// TwinCAT 3 PLC project PLC1
// ProgramVersion: 3.1.4023.0
// libraries:
//   Tc2_Standard, * (Beckhoff Automation GmbH)
//   Tc2_System, * (Beckhoff Automation GmbH)
//   Tc2_Utilities, * (Beckhoff Automation GmbH)
//   Tc3_EventLogger, * (Beckhoff Automation GmbH)
//   Tc3_Module, * (Beckhoff Automation GmbH)
//   Alarms Library,0.1,Atlantis
//   EASME Library Files,0.1,Atlantis
//   VisuSymbols,3.5.10.0,System
// project tree:
//   Alarm System/DUTs/02_Pitch/Hydair Data/ E_HydairState.TcDUT (not stored), E_LATState.TcDUT (not stored), E_MainState.TcDUT, Hydair_Data_Rcv.TcDUT (not stored), Hydair_Data_Send.TcDUT, Hydair_Ram_DataType.TcDUT (not stored), J1939_Inputs.TcDUT, J1939_outputs.TcDUT, ST_LoadSysCtrl.TcDUT (not stored), VARTYPE_EXTCANQUEUE.TcDUT
//   Alarm System/DUTs/02_Pitch/ PLCStruct.TcDUT (not stored), stLoadData.TcDUT, ST_BladePositionsEncoder.TcDUT (not stored), ST_DataSetEntry.TcDUT (not stored)
//   Alarm System/DUTs/02_Pitch/Test Rig/ E_StreamState.TcDUT (not stored)
//   Alarm System/DUTs/A. Operation_Ver2.10/02_Alarm_Handling/Alarms/ E_AlarmGroups.TcDUT, E_AlarmNames.TcDUT (not stored), E_AlarmProgram.TcDUT, E_AlarmState.TcDUT (not stored), E_BrakeProgram.TcDUT (not stored), E_ResetMode.TcDUT, ST_AlarmStructure.TcDUT, ST_Alarm_State.TcDUT (not stored), ST_Alarm_State_Alias.TcDUT (not stored), ST_AliasAlarms.TcDUT, ST_ProcessVariables.TcDUT, ST_Repetition.TcDUT (not stored), ST_RepetitionArray.TcDUT (not stored)
//   Alarm System/DUTs/A. Operation_Ver2.10/02_Alarm_Handling/StausCodes/03   STATUSCODES/ ARR_ListOfStatuscodesToBeSent.TcDUT
//   Alarm System/DUTs/A. Operation_Ver2.10/02_Alarm_Handling/StausCodes/08  Logging %28Harddisk%29/_01  Status Logger Objects/Intern/ E_FileState_SC.TcDUT (not stored), ST_FileSetup_SC.TcDUT (not stored)
//   Alarm System/DUTs/A. Operation_Ver2.10/02_Alarm_Handling/StausCodes/08  Logging %28Harddisk%29/_02  Event Logger/Logger Objects/ E_DataType.TcDUT (not stored)
//   Alarm System/DUTs/ E_IniNames.TcDUT, E_PitchState.TcDUT (not stored), stSSB_TCSInterface.TcDUT (not stored), ST_EmailSend.TcDUT (not stored), ST_EP9224_in.TcDUT (not stored), ST_EP9224_InputChannel.TcDUT, ST_EP9224_InputDevice.TcDUT (not stored), ST_EP9224_out.TcDUT, ST_EP9224_OutputChannel.TcDUT (not stored), ST_EP9224_SlaveIn.TcDUT, ST_EP9224_SlaveOut.TcDUT
//   Alarm System/DUTs/Safety/ ST_SafetyGroupData.TcDUT (not stored), ST_SafetyGroupTag.TcDUT
//   Alarm System/GVLs/A. Operation/01_General/ AlarmArrays.TcGVL, ArrIni.TcGVL (not stored), ArrLastAlarms.TcGVL (not stored), GlobVar_GeneralLog_Privat.TcGVL, GlobVar_GeneralLog_Public.TcGVL (not stored), GlobVar_LibStatuscodeLogger_Privat.TcGVL, GlobVar_ToBeReplaced_Public.TcGVL (not stored), GVL_Static.TcGVL, Operation.TcGVL (not stored), ProgramVersions.TcGVL, TurbineData.TcGVL
//   Alarm System/GVLs/A. Operation/ Global_Variables.TcGVL (not stored)
//   Alarm System/GVLs/ GVL_EventLogger.TcGVL
//   Alarm System/POUs/02_Alarm_Handling/ FB_AlarmHandler.TcPOU, FB_AlarmResetAccessCtrl.TcPOU (excluded from build), FB_AlarmResets.TcPOU, FB_AnalogueAlarm.TcPOU, FB_BrakeProgPriority.TcPOU (not stored), FB_HeaderForLogging.TcPOU (excluded from build), FB_MakeLoggString.TcPOU (excluded from build), FB_SendEmail.TcPOU, FB_StatusCodeLogger.TcPOU (excluded from build), FB_WriteEventData.TcPOU (excluded from build), FB_WriteEventData_Day.TcPOU (excluded from build), PRG_MAIN_StatuscodeLogger.TcPOU (excluded from build), PRG_Systemtime.TcPOU (not stored), P_AlarmHandling.TcPOU, P_AlarmTable.TcPOU, P_MainStatesAlarmCtrl.TcPOU (not stored), P_ScadaAlarmsMapping.TcPOU
//   Alarm System/POUs/02_Alarm_Handling/StatusCodes/ MAIN_R.TcPOU (not stored), PRG_TranslatorVarNames.TcPOU
//   Alarm System/TC3 EventLogger/ AlarmWithCustomSourceInfo.TcPOU (excluded from build), MultipleAlarmCreation.TcPOU, OtherAlarmsWithCustomSource.TcPOU (excluded from build), P_EventLogger_TCSAlarms.TcPOU
//   Base/Devices/DUT/ stError_VFD.TcDUT, stHMIMotorisedCB.TcDUT
//   Base/Devices/POU/ fbMotorisedCB.TcPOU
//   Base/Example/GVL/ GVL_HMI.TcGVL
//   Base/Example/POU/ POU_TestBase.TcPOU
//   Base/General Control/POU/ FB_AlarmEventSet.TcPOU, FB_TagAlarmProps.TcPOU, FB_Interlock.TcPOU, FB_Permissive.TcPOU, FB_SystemRunControl.TcPOU
//   Base/IO/DUT/ stError_AnalogueInput.TcDUT, stError_AnalogueOutput.TcDUT, stHMI_AnalogueInput.TcDUT, stHMI_AnalogueOutput.TcDUT, stHMI_DigitalInput.TcDUT (not stored), stHMI_DigitalOutput.TcDUT, stIOSensorTypes.TcDUT
//   Base/IO/POU/ fbIO_AnalogueInput.TcPOU, fbIO_AnalogueOutput.TcPOU, fbIO_DigitalInput.TcPOU, fbIO_DigitalOutput.TcPOU
//   Base/General Control/DUT/ stHMI_Interlock.TcDUT, stHMI_Permissive.TcDUT (not stored), stHMI_SystemRunControl.TcDUT
//   Base/Process Control/DUT/ stStep.TcDUT (not stored)
//   Base/Process Control/POU/ fb1dLookup.TcPOU, fb2dLookup.TcPOU, fbPulser.TcPOU, fbRateCalc.TcPOU, fbStepSequencer.TcPOU, POU.TcPOU
//   Base/Resource/ fbHMIBit.TcPOU
//   Base/Valve Control/DUT/ stError_Valve.TcDUT, stHMI_ValveControl.TcDUT
//   Base/Valve Control/POU/ fbValve_Solenoid.TcPOU, fcHMIBit.TcPOU
//   / GlobalTextList.TcGTLO, MAIN.TcPOU, PlcTask.TcTTO, Visualization Manager.TcVMO (not stored)
//   VISUs/ Visualization.TcVIS, Vis_AnalogueOutput_Symbol.TcVIS, Vis_DigitalInput_1.TcVIS, Vis_DigitalInput_2.TcVIS, Vis_Interlock_base.TcVIS
// real-time tasks:
//   TASK PlcTask: cycle T#10ms, priority 20, ADS port 350

CONFIGURATION PLC1
    RESOURCE PLC ON TwinCAT3
        TASK PlcTask(INTERVAL := T#10ms, PRIORITY := 20);
        PROGRAM MAIN WITH PlcTask : MAIN;
    END_RESOURCE
END_CONFIGURATION

// ---- Alarm System/DUTs/02_Pitch/Hydair Data/E_MainState.TcDUT
TYPE E_MainState :		//Is this the machine main state or the Hydraulics system??
(
	STOP:=0,
	STARTING_HYDRAULICS:=1,
	HYDRAULICS_READY:=2,
	IN_OPERATION:=3,
	PASSIVE:=5,
	MANUAL:=6,
	SAFETY_TRIPPED:=7,
	SHUTDOWN:=8
);
END_TYPE

// ---- Alarm System/DUTs/02_Pitch/Hydair Data/Hydair_Data_Send.TcDUT
TYPE Hydair_Data_Send :
STRUCT
	rRam1_LoadDemand:REAL;
	rRam2_LoadDemand:REAL;

	uiLoadsControl:ST_LoadSysCtrl;
END_STRUCT
END_TYPE

// ---- Alarm System/DUTs/02_Pitch/Hydair Data/J1939_Inputs.TcDUT
TYPE J1939_Inputs :
STRUCT
	TxCounter  : UINT;
	RxCounter  : UINT;
	NoOfRxMessages   : UINT;
	RxMessage  : ARRAY [0..11] OF VARTYPE_EXTCANQUEUE;
(*	NodeState  : USINT;
	DiagFlag   : BOOL;*)
END_STRUCT
END_TYPE

// ---- Alarm System/DUTs/02_Pitch/Hydair Data/J1939_outputs.TcDUT
TYPE J1939_outputs :
STRUCT
	TxCounter : UINT;
	RxCounter   : UINT;
	NoOfTxMessages    : UINT;
	TxMessage  : ARRAY [0..1] OF VARTYPE_EXTCANQUEUE;
END_STRUCT
END_TYPE

// ---- Alarm System/DUTs/02_Pitch/Hydair Data/VARTYPE_EXTCANQUEUE.TcDUT
TYPE VARTYPE_EXTCANQUEUE:
STRUCT
	length: UINT;
	cobId: UDINT;
	rxData: ARRAY [0..7] OF USINT;
END_STRUCT
END_TYPE

// ---- Alarm System/DUTs/02_Pitch/stLoadData.TcDUT
TYPE stLoadData :
STRUCT
	sLoadID: STRING[30];
	rRig1_LoadDemand:REAL;
	rRig2_LoadDemand:REAL;
	rRig3_LoadDemand:REAL;
	rPitchAngleDemand:REAL;
	bStart:BOOL;
	bConnect:BOOL;
	bHeartbeat:BOOL;
END_STRUCT
END_TYPE

// ---- Alarm System/DUTs/A. Operation_Ver2.10/02_Alarm_Handling/Alarms/E_AlarmGroups.TcDUT
TYPE E_AlarmGroups :
(
	Operation := 1,
	Safety := 2,
	Converter := 3,
	Pitch := 4,
	Yaw := 5,
	Nacelle := 6,
	Generator := 7,
	Gearbox := 8,
	AuxPower := 9,
	Grid := 10,
	SCADA := 11,
	BearingLube := 12,
	SealLube := 13,
	WaterMgt := 14,
	Brake := 15
);
END_TYPE

// ---- Alarm System/DUTs/A. Operation_Ver2.10/02_Alarm_Handling/Alarms/E_AlarmProgram.TcDUT
TYPE E_AlarmProgram :
(
	NoAction			:=0,	(* Prg1 *)
	Email				:=1,	(* Prg2 *)
	SMS					:=2

);
END_TYPE

// ---- Alarm System/DUTs/A. Operation_Ver2.10/02_Alarm_Handling/Alarms/E_ResetMode.TcDUT
TYPE E_ResetMode :
(
	AUTO			:=0,	(* Automatic after delay *)
	MANU			:=1	(* Manual *)
);
END_TYPE

// ---- Alarm System/DUTs/A. Operation_Ver2.10/02_Alarm_Handling/Alarms/ST_AlarmStructure.TcDUT
TYPE ST_AlarmStructure :
STRUCT
	sName:STRING;
	a:BOOL;
	b:BOOL;
	Changed:BOOL;
	iGroup:INT;
	iSetDelay:DINT;					(* 100ms *)
	iSetDelayElapsed:DINT;			(* 100ms *)
	iResetDelay:DINT;				(* 100ms *)
	iResetDelayElapsed:DINT;		(*100ms*)
	eResetMode:E_ResetMode;
	eBrakeProgram:E_BrakeProgram;
	eAlarmProgram:E_AlarmProgram;
	Enable: BOOL;
	TimeOcc: TIMESTRUCT;			(* Added 040405 KKa *)
	sTimeOcc: STRING(24); (* New *)	(* Added 091130 KKa *)
	Comment:STRING(255);

	iRepetitionNumber: INT;
	iRepetitionPeriod: INT; 					(*Minutes*)
	bRepetitionLimitExceeded: BOOL;

	Param1:ST_Parameters;
	Param2:ST_Parameters;

	iState:UDINT;(* New *)		(* Alarm state Active / Acked *)
	sID:STRING(5);(* New *)
	sClearName:STRING(90);(* New *)
	Index:INT;(* New *)
	bScope:BOOL;(* New *)

	stProcessVariables:ST_ProcessVariables; (* New *)

END_STRUCT
END_TYPE

// ---- Alarm System/DUTs/A. Operation_Ver2.10/02_Alarm_Handling/Alarms/ST_AliasAlarms.TcDUT
TYPE ST_AliasAlarms :
STRUCT
	b : INT;
END_STRUCT
END_TYPE

// ---- Alarm System/DUTs/A. Operation_Ver2.10/02_Alarm_Handling/Alarms/ST_ProcessVariables.TcDUT
TYPE ST_ProcessVariables :
STRUCT
	fPower:REAL;
	fFlowSpeed:REAL;
	fGeneratorSpeed:REAL;
	fPitchAngle:REAL;
END_STRUCT
END_TYPE

// ---- Alarm System/DUTs/A. Operation_Ver2.10/02_Alarm_Handling/StausCodes/03   STATUSCODES/ARR_ListOfStatuscodesToBeSent.TcDUT
TYPE ARR_ListOfStatuscodesToBeSent :
STRUCT
	arrListOfStatuscodesToBeSent: 		ARRAY [1..50] OF STRING [120];
END_STRUCT
END_TYPE

// ---- Alarm System/DUTs/E_IniNames.TcDUT
TYPE E_IniNames :
(
ini_fOperStartUpCounterMax := 1,
ini_fAlgHeartbeatCounterLimit := 2,
ini_fConverterCompensationAngle := 3,
ini_fConverterDampingTorqueLimitFactor := 4,
ini_fConverterDrivetrainDampingFactor1 := 5,
ini_fConverterDrivetrainDampingFactor2 := 6,
ini_fConverterDrivetrainDampingFactor3 := 7,
ini_fConverterExitToStandbyTimeout := 8,
ini_fConverterHeartbeatDelayms := 9,
ini_fConverterLookupSpeedVal0 := 10,
ini_fConverterLookupSpeedVal2 := 11,
ini_fConverterLookupSpeedVal4 := 12,
ini_fConverterLookupSpeedVal6 := 13,
ini_fConverterLookupSpeedVal8 := 14,
ini_fConverterLookupTorqueVal0 := 15,
ini_fConverterLookupTorqueVal2 := 16,
ini_fConverterLookupTorqueVal4 := 17,
ini_fConverterLookupTorqueVal6 := 18,
ini_fConverterLookupTorqueVal8 := 19,
ini_fConverterMinimumSpeedToStandby := 20,
ini_fConverterReductionReleaseFrequency := 21,
ini_fConverterReductionStartFrequency := 22,
ini_fConverterReductionStopFrequency := 23,
ini_fFlowSpeedAboveRatedLUTLength := 24,
ini_fFlowSpeedBelowRatedLUTLength := 25,
ini_fFlowSpeedTransitionLUTLength := 26,
ini_fGearboxRotorSpeedMin := 27,
ini_fGenPulloutC := 28,
ini_fGenPulloutM := 29,
ini_fGenSpeedNoiseFloor := 30,
ini_fOperEbbTideHeadingSetpoint := 31,
ini_fOperFloodTideHeadingSetpoint := 32,
ini_fOperFlowCutIn := 33,
ini_fOperFlowCutOut := 34,
ini_fOperFlowRated := 35,
ini_fOperInhibitPcsStbyToProd := 36,
ini_fOperMaxRotorPosErr := 37,
ini_fOperMinGenSyncSpeedRpm := 38,
ini_fOperRatedGeneratorSpeed := 39,
ini_fOperRotorPosCtrlErrOK := 40,
ini_fOperRotorSpeedRadsToStop := 41,
ini_fOperRotorStaticSpeedErr := 42,
ini_fOperSpeedHSSDiscrepMarginRpm := 43,
ini_fOperSpeedHSStoPCSDiscrepMarginRpm := 44,
ini_fOperSpeedLSStoHSSDiscrepMarginRpm := 45,
ini_fOperSpeedNoOfTargets := 46,
ini_fOperTrundleDuration := 47,
ini_fRotorBoltPosition := 48,
ini_fRotorEncoderZeroToBlade1 := 49,
ini_fRotorGBInputShaftPickupAPosition := 50,
ini_fRotorGBInputShaftPickupBPosition := 51,
ini_fSafetyDisablePCSEStop2 := 52,
ini_fSafetyDisablePCSEStop3 := 53,
ini_fSafetyPitchToFeatherTimeLimit := 54,
ini_fSafetyRotorDecelTimeLimit := 55,
ini_fTurbineGearboxRatio := 56,
ini_fVsprFastShutdownSpeedVal0 := 57,
ini_fVsprFastShutdownSpeedVal1 := 58,
ini_fVsprFastShutdownSpeedVal2 := 59,
ini_fVsprFastShutdownSpeedVal3 := 60,
ini_fVsprFastShutdownSpeedVal4 := 61,
ini_fVsprFastShutdownTorqueVal0 := 62,
ini_fVsprFastShutdownTorqueVal1 := 63,
ini_fVsprFastShutdownTorqueVal2 := 64,
ini_fVsprFastShutdownTorqueVal3 := 65,
ini_fVsprFastShutdownTorqueVal4 := 66,
ini_fVsprGenSpeedAtSyncSpeedRequiredTime := 67,
ini_fVsprLowSpeedSyncSpeedRPM := 68,
ini_fVsprMaximumFinePitchDeg := 69,
ini_fVsprMaximumGeneratorTorque := 70,
	ini_fVsprMinimumFinePitchDeg := 71,
ini_fVsprOptimalModeGain := 72,
ini_fVsprPositiveFeatherAngleDeg := 73,
ini_fVsprSpeedSetpointRateLimitRPMpSec := 74,
ini_fVsprStartupMinimumPitchRateLimitDegPSec := 75,
ini_fVsprSteadyShaftPowerLimit := 76,
ini_fVsprSyncSpeedTolRPM := 77,
ini_fVsprTorqueLimitSpeedVal0 := 78,
ini_fVsprTorqueLimitSpeedVal1 := 79,
ini_fVsprTorqueLimitSpeedVal2 := 80,
ini_fVsprTorqueLimitSpeedVal3 := 81,
ini_fVsprTorqueLimitSpeedVal4 := 82,
ini_fVsprTorqueLimitTorqueVal0 := 83,
ini_fVsprTorqueLimitTorqueVal1 := 84,
ini_fVsprTorqueLimitTorqueVal2 := 85,
ini_fVsprTorqueLimitTorqueVal3 := 86,
ini_fVsprTorqueLimitTorqueVal4 := 87,
ini_fWaterMgtNacelleBilgeLevelDefault := 88,
ini_fWaterMgtNacelleBilgePumpOffLevel := 89,
ini_fWaterMgtNacelleBilgePumpOffTimeMin := 90,
ini_fWaterMgtNacelleBilgePumpOffTimeout := 91,
ini_fWaterMgtNacelleBilgePumpOnLevel := 92,
ini_fWaterMgtNacelleBilgePumpOnTimeout := 93
);
END_TYPE

// ---- Alarm System/DUTs/Safety/ST_SafetyGroupTag.TcDUT
TYPE ST_SafetyGroupTag :
STRUCT
	sTitle	:STRING(80);
	bOutputSAFE	:BOOL;
	bError	:BOOL;
	bRun	:BOOL;
END_STRUCT
END_TYPE

// ---- Alarm System/DUTs/ST_EP9224_InputChannel.TcDUT
TYPE ST_EP9224_InputChannel :
STRUCT
	bErrorUs 	: BOOL;
	bErrorUp 	: BOOL;
	bWarningUs	: BOOL;
	bWarningUp	: BOOL;
	bStatusUs 	: BOOL;
	bStatusUp 	: BOOL;
	bChannelError : BOOL;
	bErrorSumCurrent 	      : BOOL;
(* This takes up a bit too much space and isn't maped by LMC, so leave it for now
	nCurrentUs 		: INT;
	nCurrentUp 		: INT;
*)
END_STRUCT
END_TYPE

// ---- Alarm System/DUTs/ST_EP9224_out.TcDUT
TYPE ST_EP9224_out :
STRUCT
	stOutput : ARRAY [1..EP9224_NUM_CHANNELS] OF ST_EP9224_OutputChannel;
	bGlobalReset : BOOL;
END_STRUCT
END_TYPE

// ---- Alarm System/DUTs/ST_EP9224_SlaveIn.TcDUT
TYPE ST_EP9224_SlaveIn :
STRUCT
	nOutput	:ARRAY [1..EP9224_NUM_CHANNELS] OF BYTE;
END_STRUCT
END_TYPE

// ---- Alarm System/DUTs/ST_EP9224_SlaveOut.TcDUT
TYPE ST_EP9224_SlaveOut :
STRUCT
	nChannel :ARRAY [1..EP9224_NUM_CHANNELS] OF BYTE;
	nStatus	 :BYTE;
END_STRUCT
END_TYPE

// ---- Base/Devices/DUT/stError_VFD.TcDUT
TYPE stError_VFD :
STRUCT
	MotorProtectorTripped: BOOL; (*Motor Protector tripped*)
	LocalDisconnectOff: BOOL; (*Motor Local switch OFF*)
	ClutchTripped: BOOL; 	(*Clutch error*)
	NoContactorFeedback: BOOL; (*No feedback from motor contactor*)
	ContactorStillOn: BOOL; (*Contactor still ON*)
	NoSignalForward: BOOL; (*No SIGNAL Forward from VFD*)
	NoSignalReverse: BOOL; (*No SIGNAL Reverse from VFD*)
	MotorNotStopped: BOOL; (*Motor doesn't stop*)
	MaxFrequencyReached: BOOL; (*Max frequency reached*)
	Overcurrent: BOOL; (*VFD overcurrent*)
	MotorOverload: BOOL; (*Motor overload*)
	VFDOverload: BOOL; (*VFD overload*)
	GeneralFault: BOOL; (*VFD fault*)
	NoCoolingFanFeedback: BOOL; (*Cooling fan did not come on within 30 seconds*)
END_STRUCT
END_TYPE

// ---- Base/Devices/DUT/stHMIMotorisedCB.TcDUT
TYPE stHMIMotorisedCB :
STRUCT
	iMode: 			 INT;
	iErrorCode:		 INT;		
	iStatus	:		 INT;	
	bPB_ResetError:	 BOOL; (*Reset errors pushbutton*)
	bPBEN_ResetError:BOOL; (*Reset Error pushbutton enable*)
	bPBOpen: 		 BOOL; (*Pushbutton command open from HMI*)
	bPBClose:		 BOOL; (*Pushbutton command close from HMI*)
	bPBEN_Open:		 BOOL; (*Pushbuton enable open command from HMI*)
	bPBEN_Close: 	 BOOL; (*Pushbuton enable open command from HMI*)
	bSignalClosed:	 BOOL; (*MCB closed feedback*)
	bSignalOpened: 	 BOOL; (*MCB Opened feedback*)
	bCloseON:		 BOOL; (*Close command is ON*)
	bOpenON:		 BOOL; (*Open command is ON*)
	bError:			 BOOL; (*Error Status*)
	bInterlock: 	 BOOL;	(*MCB Interlocked*)
END_STRUCT
END_TYPE

// ---- Base/IO/DUT/stError_AnalogueInput.TcDUT
TYPE stError_AnalogueInput :
STRUCT
	LowLowAlarm:BOOL; 	(*Value below low low set point*)
	HighHighAlarm:BOOL; (*Value above high high set point*)
	Invalid:BOOL; 		(*Invalid input*)
END_STRUCT
END_TYPE

// ---- Base/IO/DUT/stError_AnalogueOutput.TcDUT
TYPE stError_AnalogueOutput :
STRUCT
	Out_Of_Range:BOOL;			//Input Value is outside range of Engineering Units
	Configuration_Error:BOOL;	//Engineering Units are not properly configured
END_STRUCT
END_TYPE

// ---- Base/IO/DUT/stHMI_AnalogueInput.TcDUT
TYPE stHMI_AnalogueInput :
STRUCT
	iMode:INT; 			(*Current mode*)
	iErrorCode: INT; 	(*Error code*)
	iStatus:INT; 		(*Overall HMI Status*)
	rActiveValue:REAL;	(* Used Value, Input OR Override*)
	rInputValue:REAL; 	(*Input Value*)
	rManualValue:REAL; 	(*Manual mode simulated value*)
	bPB_ResetError:BOOL;  (*Reset errors pushbutton*)
	bPBEN_ResetError:BOOL; (*Reset error pushbutton enabled*)
	bError:BOOL;
END_STRUCT
END_TYPE

// ---- Base/IO/DUT/stHMI_AnalogueOutput.TcDUT
TYPE stHMI_AnalogueOutput :
STRUCT
	iMode: 			INT;		//Current mode
	iErrorCode:		INT; 		//error code	
	rValue:			REAL;		//Output Value
	rManualValue:	REAL;		//Manual mode value
	rAutoValue:		REAL;		 //Auto Mode Value
	rEstopValue:	REAL;		//Estop condition custom value
	bPB_ResetError:	BOOL;		//Reset errors pushbutton
	bPBEN_ResetError:	BOOL;	//Reset error pushbutton enabled
	bError:	BOOL;				//Overall error
	bInterlock:	BOOL;	//Analogue output is interlocked
	iEstopFunction:INT;	//Enumerated value of E-Stop response constant
END_STRUCT
END_TYPE

// ---- Base/IO/DUT/stHMI_DigitalOutput.TcDUT
TYPE stHMI_DigitalOutput :
STRUCT
	iMode:INT;			(*Current mode*)
	bCommand: BOOL;		(*Output command status*)
	bCommandAuto:BOOL;	(*the output command from the PLC, ignoring manual overrides*)
	bInterlock:BOOL;	(*Digital output is interlocked*)
	bPB_On:BOOL;		(*Command on override pushbutton*)
	bPB_Off:BOOL;		(*Command off override pushbutton*)
	bPBEN_On:BOOL;		(*Command on override pushbutton enabled*)
	bPBEN_Off:BOOL;		(*Command off override pushbutton enabled*)
END_STRUCT
END_TYPE

// ---- Base/IO/DUT/stIOSensorTypes.TcDUT
{attribute 'qualified_only'}
{attribute 'strict'}
TYPE stIOSensorTypes :
(
	AI_4To20ma := 0,
	AI_PT100	:= 1,
	AI_0To10V	:=2,
	AI_0To5V	:=3
	
);
END_TYPE

// ---- Base/General Control/DUT/stHMI_Interlock.TcDUT
TYPE stHMI_Interlock :
STRUCT
	abInterlocks: ARRAY[1..16] OF BOOL;
	asInterlockNames: ARRAY[1..16] OF STRING[20];
	bInterlockOk:BOOL;
END_STRUCT
END_TYPE

// ---- Base/General Control/DUT/stHMI_SystemRunControl.TcDUT
TYPE stHMI_SystemRunControl :
STRUCT
	bRunning:BOOL; 	  (*System is running*)
	bPB_Start:BOOL;    (*Start command pushbutton*)
	bPB_Stop:BOOL;	  (*Stop command pushbutton*)
	bPBEN_Start:BOOL;  (*Start command pushbutton enable*)
	bPBEN_Stop:BOOL;  (*Stop command pushbutton enable*)
END_STRUCT
END_TYPE

// ---- Base/Valve Control/DUT/stError_Valve.TcDUT
TYPE stError_Valve :
STRUCT
	NoHomeFeedback:BOOL;			//Home position feedback not active
	NoWorkFeedback:BOOL;			//Work position feedback not active
	HomeFeedbackStillActive: BOOL;	//Home position feedback still active when commanded to Work Position
	WorkFeedbackStillActive: BOOL;	//Work position feedback still active when commanded to Home Position
END_STRUCT
END_TYPE

// ---- Base/Valve Control/DUT/stHMI_ValveControl.TcDUT
TYPE stHMI_ValveControl :
STRUCT
	iMode	:		 INT;		//Current mode				
	iErrorCode:		 INT;		//
	iStatus	:		 INT;		//
	bPB_ResetError:	 BOOL;		//Reset errors pushbutton
	bPB_Home:		 BOOL;		//Move to home in manual mode pushbutton
	bPB_Work:		 BOOL;		//Move to work in manual mode pushbutton
	bPBEN_ResetError:BOOL;		//Reset Error pushbutton enable
	bPBEN_Home:		 BOOL;		//Home pushbutton enabled
	bPBEN_Work:		 BOOL;		//Work pushbutton enabledv
	bHomeOn:		 BOOL;		//Home command is on
	bWorkOn:		 BOOL;		//Work command is on
	bSignalHome:	 BOOL;		//Home feedback
	bSignalWork:	 BOOL;		//Work feedback
	bError:			 BOOL;		//Error Status
	bInterlock: 	 BOOL;		//Valve Interlocked
END_STRUCT
END_TYPE

// ---- Alarm System/GVLs/A. Operation/01_General/AlarmArrays.TcGVL
{attribute 'Tc2GvlVarNames'}
VAR_GLOBAL
	{attribute 'OPC.UA.DA' := '1'}
	{attribute 'OPC.UA.DA.StructuredType' := '1'}
	arrScadaAlarms : ARRAY [1..222]  OF ST_AliasAlarms;	
	
	{attribute 'OPC.UA.DA' := '1'}
	{attribute 'OPC.UA.DA.StructuredType' := '1'}
	arrOPCUA_Alarms : ARRAY [1..10]  OF ST_Alarm_State_Alias;	
	
	
END_VAR


VAR_GLOBAL PERSISTENT
stOperAlarmIniFileName: STRING:='Alarms_AR2000.xls 011021';
arrAlarmsOld: ARRAY [1..222] OF ST_AlarmStructure;
arrAlarmsOriginal,arrAlarms: ARRAY [1..222] OF ST_AlarmStructure :=[
( sName := 'a_bOperMaStInitSt', sClearName := '', sID := '1001', a := FALSE, b := FALSE, iGroup :=1, iSetDelay :=0, iResetDelay := 100, eResetMode := MANU, eBrakeProgram := B100, eAlarmProgram := 0, Enable := TRUE, iRepetitionNumber := 0 , iRepetitionPeriod := 10, Comment := 'Turbine Initialising', Param1 := (Set:=0, SetMin:=0, SetMax:=0,Comment:=''), Param2 := (Set:=0, SetMin:=0, SetMax:=0,Comment:='') ),
( sName := 'a_bOperMaStStopSt', sClearName := '', sID := '1002', a := FALSE, b := FALSE, iGroup :=1, iSetDelay :=0, iResetDelay := 0, eResetMode := MANU, eBrakeProgram := B100, eAlarmProgram := 0, Enable := TRUE, iRepetitionNumber := 0 , iRepetitionPeriod := 10, Comment := 'Turbine in the Stop state', Param1 := (Set:=0, SetMin:=0, SetMax:=0,Comment:=''), Param2 := (Set:=0, SetMin:=0, SetMax:=0,Comment:='') ),
( sName := 'a_bOperMaStIdleSt', sClearName := '', sID := '1003', a := FALSE, b := FALSE, iGroup :=1, iSetDelay :=0, iResetDelay := 0, eResetMode := MANU, eBrakeProgram := B100, eAlarmProgram := 0, Enable := TRUE, iRepetitionNumber := 0 , iRepetitionPeriod := 10, Comment := 'Turbine in the Idle state', Param1 := (Set:=0, SetMin:=0, SetMax:=0,Comment:=''), Param2 := (Set:=0, SetMin:=0, SetMax:=0,Comment:='') ),
( sName := 'a_bOperMaStStandbySt', sClearName := '', sID := '1004', a := FALSE, b := FALSE, iGroup :=1, iSetDelay :=0, iResetDelay := 0, eResetMode := MANU, eBrakeProgram := B100, eAlarmProgram := 0, Enable := TRUE, iRepetitionNumber := 0 , iRepetitionPeriod := 10, Comment := 'Turbine in the Ready state', Param1 := (Set:=0, SetMin:=0, SetMax:=0,Comment:=''), Param2 := (Set:=0, SetMin:=0, SetMax:=0,Comment:='') ),
( sName := 'a_bOperMaStPowerProductionSt', sClearName := '', sID := '1005', a := FALSE, b := FALSE, iGroup :=1, iSetDelay :=0, iResetDelay := 0, eResetMode := MANU, eBrakeProgram := B100, eAlarmProgram := 0, Enable := TRUE, iRepetitionNumber := 0 , iRepetitionPeriod := 10, Comment := 'Turbine in the Power Production state', Param1 := (Set:=0, SetMin:=0, SetMax:=0,Comment:=''), Param2 := (Set:=0, SetMin:=0, SetMax:=0,Comment:='') ),
( sName := 'a_bOperMaStNormalStopSt', sClearName := '', sID := '1006', a := FALSE, b := FALSE, iGroup :=1, iSetDelay :=0, iResetDelay := 0, eResetMode := MANU, eBrakeProgram := B100, eAlarmProgram := 0, Enable := TRUE, iRepetitionNumber := 0 , iRepetitionPeriod := 10, Comment := 'Turbine in the Normal Stop state', Param1 := (Set:=0, SetMin:=0, SetMax:=0,Comment:=''), Param2 := (Set:=0, SetMin:=0, SetMax:=0,Comment:='') ),
( sName := 'a_bOperMaStEmergencyStopSt', sClearName := '', sID := '1007', a := FALSE, b := FALSE, iGroup :=1, iSetDelay :=0, iResetDelay := 0, eResetMode := MANU, eBrakeProgram := B100, eAlarmProgram := 0, Enable := TRUE, iRepetitionNumber := 0 , iRepetitionPeriod := 10, Comment := 'Turbine in the Emergency Stop state', Param1 := (Set:=0, SetMin:=0, SetMax:=0,Comment:=''), Param2 := (Set:=0, SetMin:=0, SetMax:=0,Comment:='') ),
( sName := 'a_bOperAutostartCmdActive', sClearName := '', sID := '1008', a := FALSE, b := FALSE, iGroup :=1, iSetDelay :=0, iResetDelay := 0, eResetMode := MANU, eBrakeProgram := B99, eAlarmProgram := 0, Enable := TRUE, iRepetitionNumber := 0 , iRepetitionPeriod := 0, Comment := 'System generation inhibit removed by operator', Param1 := (Set:=0, SetMin:=0, SetMax:=0,Comment:=''), Param2 := (Set:=0, SetMin:=0, SetMax:=0,Comment:='') ),
( sName := 'a_bOperTestIdlingShutdown', sClearName := '', sID := '1009', a := FALSE, b := FALSE, iGroup :=1, iSetDelay :=0, iResetDelay := 0, eResetMode := MANU, eBrakeProgram := B17, eAlarmProgram := 0, Enable := TRUE, iRepetitionNumber := 0 , iRepetitionPeriod := 0, Comment := 'Test B17 go to Idle or Standby', Param1 := (Set:=0, SetMin:=0, SetMax:=0,Comment:=''), Param2 := (Set:=0, SetMin:=0, SetMax:=0,Comment:='') ),
( sName := 'a_bOperTestBrakingShutdown', sClearName := '', sID := '1010', a := FALSE, b := FALSE, iGroup :=1, iSetDelay :=0, iResetDelay := 0, eResetMode := MANU, eBrakeProgram := B14, eAlarmProgram := 0, Enable := TRUE, iRepetitionNumber := 0 , iRepetitionPeriod := 0, Comment := 'Test B14 apply parking brake', Param1 := (Set:=0, SetMin:=0, SetMax:=0,Comment:=''), Param2 := (Set:=0, SetMin:=0, SetMax:=0,Comment:='') ),
( sName := 'a_bOperTestSafetyVCTripShutdown', sClearName := '', sID := '1011', a := FALSE, b := FALSE, iGroup :=1, iSetDelay :=0, iResetDelay := 0, eResetMode := MANU, eBrakeProgram := B100, eAlarmProgram := 0, Enable := TRUE, iRepetitionNumber := 0 , iRepetitionPeriod := 0, Comment := 'Test B9 trip vacuum contactor', Param1 := (Set:=0, SetMin:=0, SetMax:=0,Comment:=''), Param2 := (Set:=0, SetMin:=0, SetMax:=0,Comment:='') ),
( sName := 'a_bOperTestSafetyBrakeShutdown', sClearName := '', sID := '1012', a := FALSE, b := FALSE, iGroup :=1, iSetDelay :=0, iResetDelay := 0, eResetMode := MANU, eBrakeProgram := B100, eAlarmProgram := 0, Enable := TRUE, iRepetitionNumber := 0 , iRepetitionPeriod := 0, Comment := 'Test B5 apply safety brake', Param1 := (Set:=0, SetMin:=0, SetMax:=0,Comment:=''), Param2 := (Set:=0, SetMin:=0, SetMax:=0,Comment:='') ),
( sName := 'a_bOperCmdNormalShutdownToStop', sClearName := 'Turbine manual stop using main gui button', sID := '1013', a := FALSE, b := FALSE, iGroup :=1, iSetDelay :=0, iResetDelay := 0, eResetMode := MANU, eBrakeProgram := B100, eAlarmProgram := 0, Enable := TRUE, iRepetitionNumber := 0 , iRepetitionPeriod := 0, Comment := 'Manual stop command', Param1 := (Set:=0, SetMin:=0, SetMax:=0,Comment:=''), Param2 := (Set:=0, SetMin:=0, SetMax:=0,Comment:='') ),
( sName := 'a_bOperCmdNormalShutdownToStandby', sClearName := '', sID := '1014', a := FALSE, b := FALSE, iGroup :=1, iSetDelay :=0, iResetDelay := 0, eResetMode := MANU, eBrakeProgram := B100, eAlarmProgram := 0, Enable := TRUE, iRepetitionNumber := 0 , iRepetitionPeriod := 0, Comment := '', Param1 := (Set:=0, SetMin:=0, SetMax:=0,Comment:=''), Param2 := (Set:=0, SetMin:=0, SetMax:=0,Comment:='') ),
( sName := 'a_bOperRepeatingAlarm', sClearName := '', sID := '1015', a := FALSE, b := FALSE, iGroup :=1, iSetDelay :=10, iResetDelay := 0, eResetMode := MANU, eBrakeProgram := B100, eAlarmProgram := 0, Enable := TRUE, iRepetitionNumber := 0 , iRepetitionPeriod := 10, Comment := 'Alarm which occur with this one has occured too many times', Param1 := (Set:=0, SetMin:=0, SetMax:=0,Comment:=''), Param2 := (Set:=0, SetMin:=0, SetMax:=0,Comment:='') ),
( sName := 'a_bOperResetTooLongPushed', sClearName := 'Reset Button ', sID := '1016', a := FALSE, b := FALSE, iGroup :=1, iSetDelay :=10, iResetDelay := 0, eResetMode := MANU, eBrakeProgram := B99, eAlarmProgram := 0, Enable := TRUE, iRepetitionNumber := 0 , iRepetitionPeriod := 10, Comment := 'Reset button pressed too long', Param1 := (Set:=0, SetMin:=0, SetMax:=0,Comment:=''), Param2 := (Set:=0, SetMin:=0, SetMax:=0,Comment:='') ),
( sName := 'a_bOperAlarmParameterChanged', sClearName := 'Alarm Parameter ', sID := '1017', a := FALSE, b := FALSE, iGroup :=1, iSetDelay :=0, iResetDelay := 5, eResetMode := MANU, eBrakeProgram := B99, eAlarmProgram := 0, Enable := TRUE, iRepetitionNumber := 0 , iRepetitionPeriod := 10, Comment := 'Alarm parameter has been changed', Param1 := (Set:=0, SetMin:=0, SetMax:=0,Comment:=''), Param2 := (Set:=0, SetMin:=0, SetMax:=0,Comment:='') ),
( sName := 'a_bOperIniParameterChanged', sClearName := 'Ini Parameter ', sID := '1018', a := FALSE, b := FALSE, iGroup :=1, iSetDelay :=0, iResetDelay := 5, eResetMode := MANU, eBrakeProgram := B99, eAlarmProgram := 0, Enable := TRUE, iRepetitionNumber := 0 , iRepetitionPeriod := 10, Comment := 'Ini parameter has been changed', Param1 := (Set:=0, SetMin:=0, SetMax:=0,Comment:=''), Param2 := (Set:=0, SetMin:=0, SetMax:=0,Comment:='') ),
( sName := 'a_bOperSystemReboot', sClearName := 'System ', sID := '1019', a := FALSE, b := FALSE, iGroup :=1, iSetDelay :=10, iResetDelay := 150, eResetMode := MANU, eBrakeProgram := B100, eAlarmProgram := 0, Enable := TRUE, iRepetitionNumber := 0 , iRepetitionPeriod := 10, Comment := 'System is rebooted', Param1 := (Set:=0, SetMin:=0, SetMax:=0,Comment:=''), Param2 := (Set:=0, SetMin:=0, SetMax:=0,Comment:='') ),
( sName := 'a_bOperSystemRestart ', sClearName := 'System ', sID := '1020', a := FALSE, b := FALSE, iGroup :=1, iSetDelay :=10, iResetDelay := 150, eResetMode := MANU, eBrakeProgram := B100, eAlarmProgram := 0, Enable := TRUE, iRepetitionNumber := 0 , iRepetitionPeriod := 10, Comment := 'System is restarted', Param1 := (Set:=0, SetMin:=0, SetMax:=0,Comment:=''), Param2 := (Set:=0, SetMin:=0, SetMax:=0,Comment:='') ),
( sName := 'a_bOperScopeViewNotActive', sClearName := 'ScopeView running', sID := '1021', a := FALSE, b := FALSE, iGroup :=1, iSetDelay :=100, iResetDelay := 0, eResetMode := MANU, eBrakeProgram := B17, eAlarmProgram := 0, Enable := TRUE, iRepetitionNumber := 0 , iRepetitionPeriod := 10, Comment := 'Fastlog system not active', Param1 := (Set:=0, SetMin:=0, SetMax:=0,Comment:=''), Param2 := (Set:=0, SetMin:=0, SetMax:=0,Comment:='') ),
( sName := 'a_bOperXMLDataUncertainty', sClearName := 'Turbine data XML file Ok', sID := '1022', a := FALSE, b := FALSE, iGroup :=1, iSetDelay :=0, iResetDelay := 0, eResetMode := MANU, eBrakeProgram := B17, eAlarmProgram := 0, Enable := TRUE, iRepetitionNumber := 0 , iRepetitionPeriod := 10, Comment := 'Turbine data XML file uncertainty', Param1 := (Set:=0, SetMin:=0, SetMax:=0,Comment:=''), Param2 := (Set:=0, SetMin:=0, SetMax:=0,Comment:='') ),
( sName := 'a_bOperSoftwareUpdate', sClearName := 'System software ', sID := '1023', a := FALSE, b := FALSE, iGroup :=1, iSetDelay :=0, iResetDelay := 0, eResetMode := MANU, eBrakeProgram := B17, eAlarmProgram := 0, Enable := FALSE, iRepetitionNumber := 0 , iRepetitionPeriod := 10, Comment := 'System software is updated', Param1 := (Set:=0, SetMin:=0, SetMax:=0,Comment:=''), Param2 := (Set:=0, SetMin:=0, SetMax:=0,Comment:='') ),
( sName := 'a_bOperFastlogComsErr', sClearName := 'a_bOperLossOfCommsToArrayController', sID := '1024', a := FALSE, b := FALSE, iGroup :=1, iSetDelay :=0, iResetDelay := 0, eResetMode := MANU, eBrakeProgram := B99, eAlarmProgram := 0, Enable := TRUE, iRepetitionNumber := 0 , iRepetitionPeriod := 10, Comment := 'Loss of Comms with ARL Array PLC', Param1 := (Set:=0, SetMin:=0, SetMax:=0,Comment:=''), Param2 := (Set:=0, SetMin:=0, SetMax:=0,Comment:='') ),
( sName := 'a_bOperInOffMode', sClearName := 'Turbine in OFF Mode', sID := '1025', a := FALSE, b := FALSE, iGroup :=1, iSetDelay :=0, iResetDelay := 0, eResetMode := MANU, eBrakeProgram := B100, eAlarmProgram := 0, Enable := TRUE, iRepetitionNumber := 0 , iRepetitionPeriod := 10, Comment := 'Turbine entering OFF Mode', Param1 := (Set:=0, SetMin:=0, SetMax:=0,Comment:=''), Param2 := (Set:=0, SetMin:=0, SetMax:=0,Comment:='') ),
( sName := 'a_bOperInServiceMode', sClearName := 'Turbine in Service Mode', sID := '1026', a := FALSE, b := FALSE, iGroup :=1, iSetDelay :=0, iResetDelay := 0, eResetMode := MANU, eBrakeProgram := B100, eAlarmProgram := 0, Enable := TRUE, iRepetitionNumber := 0 , iRepetitionPeriod := 10, Comment := 'Turbine entering Service Mode', Param1 := (Set:=0, SetMin:=0, SetMax:=0,Comment:=''), Param2 := (Set:=0, SetMin:=0, SetMax:=0,Comment:='') ),
( sName := 'a_bOperInAutomaticMode', sClearName := 'Turbine in Automatic Mode', sID := '1027', a := FALSE, b := FALSE, iGroup :=1, iSetDelay :=0, iResetDelay := 0, eResetMode := MANU, eBrakeProgram := B100, eAlarmProgram := 0, Enable := TRUE, iRepetitionNumber := 0 , iRepetitionPeriod := 10, Comment := 'Turbine entering Automatic Mode', Param1 := (Set:=0, SetMin:=0, SetMax:=0,Comment:=''), Param2 := (Set:=0, SetMin:=0, SetMax:=0,Comment:='') ),
( sName := 'a_bOperInManualMode', sClearName := 'Turbine in Manual Mode', sID := '1028', a := FALSE, b := FALSE, iGroup :=1, iSetDelay :=0, iResetDelay := 0, eResetMode := MANU, eBrakeProgram := B100, eAlarmProgram := 0, Enable := TRUE, iRepetitionNumber := 0 , iRepetitionPeriod := 10, Comment := 'Turbine entering Manual Mode', Param1 := (Set:=0, SetMin:=0, SetMax:=0,Comment:=''), Param2 := (Set:=0, SetMin:=0, SetMax:=0,Comment:='') ),
( sName := 'a_bOperInFATMode', sClearName := 'Turbine in Factory Acceptance Test Nautilus Mode', sID := '1029', a := FALSE, b := FALSE, iGroup :=1, iSetDelay :=0, iResetDelay := 0, eResetMode := MANU, eBrakeProgram := B100, eAlarmProgram := 0, Enable := TRUE, iRepetitionNumber := 0 , iRepetitionPeriod := 10, Comment := 'Turbine entering Factory Acceptance Test Nautilus Mode', Param1 := (Set:=0, SetMin:=0, SetMax:=0,Comment:=''), Param2 := (Set:=0, SetMin:=0, SetMax:=0,Comment:='') ),
( sName := 'a_bHydairFaultActive', sClearName := 'Cleared', sID := '1030', a := FALSE, b := FALSE, iGroup :=1, iSetDelay :=0, iResetDelay := 0, eResetMode := MANU, eBrakeProgram := B99, eAlarmProgram := 0, Enable := TRUE, iRepetitionNumber := 0 , iRepetitionPeriod := 0, Comment := '', Param1 := (Set:=0, SetMin:=0, SetMax:=0,Comment:=''), Param2 := (Set:=0, SetMin:=0, SetMax:=0,Comment:='') ),
( sName := 'a_bHydairOfflineFilterClogged', sClearName := 'Cleared', sID := '1031', a := FALSE, b := FALSE, iGroup :=1, iSetDelay :=0, iResetDelay := 0, eResetMode := MANU, eBrakeProgram := B99, eAlarmProgram := 0, Enable := TRUE, iRepetitionNumber := 0 , iRepetitionPeriod := 0, Comment := '', Param1 := (Set:=0, SetMin:=0, SetMax:=0,Comment:=''), Param2 := (Set:=0, SetMin:=0, SetMax:=0,Comment:='') ),
( sName := 'a_bMainReturnPressureFilterClogged', sClearName := 'Cleared', sID := '1032', a := FALSE, b := FALSE, iGroup :=1, iSetDelay :=0, iResetDelay := 0, eResetMode := MANU, eBrakeProgram := B99, eAlarmProgram := 0, Enable := TRUE, iRepetitionNumber := 0 , iRepetitionPeriod := 0, Comment := '', Param1 := (Set:=0, SetMin:=0, SetMax:=0,Comment:=''), Param2 := (Set:=0, SetMin:=0, SetMax:=0,Comment:='') ),
( sName := 'a_bMainSupplyPressureFilterClogged', sClearName := 'Cleared', sID := '1033', a := FALSE, b := FALSE, iGroup :=1, iSetDelay :=0, iResetDelay := 0, eResetMode := MANU, eBrakeProgram := B99, eAlarmProgram := 0, Enable := TRUE, iRepetitionNumber := 0 , iRepetitionPeriod := 0, Comment := '', Param1 := (Set:=0, SetMin:=0, SetMax:=0,Comment:=''), Param2 := (Set:=0, SetMin:=0, SetMax:=0,Comment:='') ),
( sName := 'a_bHydairPassiveCtrlState', sClearName := 'Cleared', sID := '1034', a := FALSE, b := FALSE, iGroup :=1, iSetDelay :=0, iResetDelay := 0, eResetMode := MANU, eBrakeProgram := B99, eAlarmProgram := 0, Enable := TRUE, iRepetitionNumber := 0 , iRepetitionPeriod := 0, Comment := '', Param1 := (Set:=0, SetMin:=0, SetMax:=0,Comment:=''), Param2 := (Set:=0, SetMin:=0, SetMax:=0,Comment:='') ),
( sName := 'a_bHydairStartUp', sClearName := 'Cleared', sID := '1035', a := FALSE, b := FALSE, iGroup :=1, iSetDelay :=0, iResetDelay := 0, eResetMode := MANU, eBrakeProgram := B99, eAlarmProgram := 0, Enable := TRUE, iRepetitionNumber := 0 , iRepetitionPeriod := 0, Comment := '', Param1 := (Set:=0, SetMin:=0, SetMax:=0,Comment:=''), Param2 := (Set:=0, SetMin:=0, SetMax:=0,Comment:='') ),
( sName := 'a_bHydairReadyToOperate', sClearName := 'Cleared', sID := '1036', a := FALSE, b := FALSE, iGroup :=1, iSetDelay :=0, iResetDelay := 0, eResetMode := MANU, eBrakeProgram := B99, eAlarmProgram := 0, Enable := TRUE, iRepetitionNumber := 0 , iRepetitionPeriod := 0, Comment := '', Param1 := (Set:=0, SetMin:=0, SetMax:=0,Comment:=''), Param2 := (Set:=0, SetMin:=0, SetMax:=0,Comment:='') ),
( sName := 'a_bHydairActiveCtrlState', sClearName := 'Cleared', sID := '1037', a := FALSE, b := FALSE, iGroup :=1, iSetDelay :=0, iResetDelay := 0, eResetMode := MANU, eBrakeProgram := B99, eAlarmProgram := 0, Enable := TRUE, iRepetitionNumber := 0 , iRepetitionPeriod := 0, Comment := '', Param1 := (Set:=0, SetMin:=0, SetMax:=0,Comment:=''), Param2 := (Set:=0, SetMin:=0, SetMax:=0,Comment:='') ),
( sName := 'a_bHydairStopped', sClearName := 'Cleared', sID := '1038', a := FALSE, b := FALSE, iGroup :=1, iSetDelay :=0, iResetDelay := 0, eResetMode := MANU, eBrakeProgram := B99, eAlarmProgram := 0, Enable := TRUE, iRepetitionNumber := 0 , iRepetitionPeriod := 0, Comment := '', Param1 := (Set:=0, SetMin:=0, SetMax:=0,Comment:=''), Param2 := (Set:=0, SetMin:=0, SetMax:=0,Comment:='') ),
( sName := 'a_bHydairEstopActive', sClearName := 'Cleared', sID := '1039', a := FALSE, b := FALSE, iGroup :=1, iSetDelay :=0, iResetDelay := 0, eResetMode := MANU, eBrakeProgram := B99, eAlarmProgram := 0, Enable := TRUE, iRepetitionNumber := 0 , iRepetitionPeriod := 0, Comment := '', Param1 := (Set:=0, SetMin:=0, SetMax:=0,Comment:=''), Param2 := (Set:=0, SetMin:=0, SetMax:=0,Comment:='') ),
( sName := 'a_bHydairOilTempTooHigh', sClearName := 'Cleared', sID := '1040', a := FALSE, b := FALSE, iGroup :=1, iSetDelay :=0, iResetDelay := 0, eResetMode := MANU, eBrakeProgram := B99, eAlarmProgram := 0, Enable := TRUE, iRepetitionNumber := 0 , iRepetitionPeriod := 0, Comment := '', Param1 := (Set:=0, SetMin:=0, SetMax:=0,Comment:=''), Param2 := (Set:=0, SetMin:=0, SetMax:=0,Comment:='') ),
( sName := 'a_bHydairReadyToStartup', sClearName := 'Cleared', sID := '1041', a := FALSE, b := FALSE, iGroup :=1, iSetDelay :=0, iResetDelay := 0, eResetMode := MANU, eBrakeProgram := B99, eAlarmProgram := 0, Enable := TRUE, iRepetitionNumber := 0 , iRepetitionPeriod := 0, Comment := '', Param1 := (Set:=0, SetMin:=0, SetMax:=0,Comment:=''), Param2 := (Set:=0, SetMin:=0, SetMax:=0,Comment:='') ),
( sName := 'a_bOperRequestStopLATSystem', sClearName := 'Cleared', sID := '1042', a := FALSE, b := FALSE, iGroup :=1, iSetDelay :=0, iResetDelay := 0, eResetMode := MANU, eBrakeProgram := B99, eAlarmProgram := 0, Enable := TRUE, iRepetitionNumber := 0 , iRepetitionPeriod := 0, Comment := '', Param1 := (Set:=0, SetMin:=0, SetMax:=0,Comment:=''), Param2 := (Set:=0, SetMin:=0, SetMax:=0,Comment:='') ),
( sName := 'a_bOperRequestStartupHydair', sClearName := 'Cleared', sID := '1043', a := FALSE, b := FALSE, iGroup :=1, iSetDelay :=0, iResetDelay := 0, eResetMode := MANU, eBrakeProgram := B99, eAlarmProgram := 0, Enable := TRUE, iRepetitionNumber := 0 , iRepetitionPeriod := 0, Comment := '', Param1 := (Set:=0, SetMin:=0, SetMax:=0,Comment:=''), Param2 := (Set:=0, SetMin:=0, SetMax:=0,Comment:='') ),
( sName := 'a_bOperRequestPassivePitchCtrl', sClearName := 'Cleared', sID := '1044', a := FALSE, b := FALSE, iGroup :=1, iSetDelay :=0, iResetDelay := 0, eResetMode := MANU, eBrakeProgram := B99, eAlarmProgram := 0, Enable := TRUE, iRepetitionNumber := 0 , iRepetitionPeriod := 0, Comment := '', Param1 := (Set:=0, SetMin:=0, SetMax:=0,Comment:=''), Param2 := (Set:=0, SetMin:=0, SetMax:=0,Comment:='') ),
( sName := 'a_bOperRequestActiveLoadCtrlMode', sClearName := 'Cleared', sID := '1045', a := FALSE, b := FALSE, iGroup :=1, iSetDelay :=0, iResetDelay := 0, eResetMode := MANU, eBrakeProgram := B99, eAlarmProgram := 0, Enable := TRUE, iRepetitionNumber := 0 , iRepetitionPeriod := 0, Comment := '', Param1 := (Set:=0, SetMin:=0, SetMax:=0,Comment:=''), Param2 := (Set:=0, SetMin:=0, SetMax:=0,Comment:='') ),
( sName := 'a_bOperRequestLoadProfileStream', sClearName := 'Cleared', sID := '1046', a := FALSE, b := FALSE, iGroup :=1, iSetDelay :=0, iResetDelay := 0, eResetMode := MANU, eBrakeProgram := B99, eAlarmProgram := 0, Enable := TRUE, iRepetitionNumber := 0 , iRepetitionPeriod := 0, Comment := '', Param1 := (Set:=0, SetMin:=0, SetMax:=0,Comment:=''), Param2 := (Set:=0, SetMin:=0, SetMax:=0,Comment:='') ),
( sName := 'a_bOperLoadProfileStreamingStarted', sClearName := 'Cleared', sID := '1047', a := FALSE, b := FALSE, iGroup :=1, iSetDelay :=0, iResetDelay := 0, eResetMode := MANU, eBrakeProgram := B99, eAlarmProgram := 0, Enable := TRUE, iRepetitionNumber := 0 , iRepetitionPeriod := 0, Comment := '', Param1 := (Set:=0, SetMin:=0, SetMax:=0,Comment:=''), Param2 := (Set:=0, SetMin:=0, SetMax:=0,Comment:='') ),
( sName := 'a_bOperLoadProfilePaused', sClearName := 'Cleared', sID := '1048', a := FALSE, b := FALSE, iGroup :=1, iSetDelay :=0, iResetDelay := 0, eResetMode := MANU, eBrakeProgram := B99, eAlarmProgram := 0, Enable := TRUE, iRepetitionNumber := 0 , iRepetitionPeriod := 0, Comment := '', Param1 := (Set:=0, SetMin:=0, SetMax:=0,Comment:=''), Param2 := (Set:=0, SetMin:=0, SetMax:=0,Comment:='') ),
( sName := 'a_bOperLoadProfileFrequencyError', sClearName := 'Cleared', sID := '1049', a := FALSE, b := FALSE, iGroup :=1, iSetDelay :=0, iResetDelay := 0, eResetMode := MANU, eBrakeProgram := B99, eAlarmProgram := 0, Enable := TRUE, iRepetitionNumber := 0 , iRepetitionPeriod := 0, Comment := '', Param1 := (Set:=0, SetMin:=0, SetMax:=0,Comment:=''), Param2 := (Set:=0, SetMin:=0, SetMax:=0,Comment:='') ),
( sName := 'a_bOperPitch100HrRuntime', sClearName := 'Cleared', sID := '1050', a := FALSE, b := FALSE, iGroup :=1, iSetDelay :=0, iResetDelay := 0, eResetMode := MANU, eBrakeProgram := B99, eAlarmProgram := 0, Enable := TRUE, iRepetitionNumber := 0 , iRepetitionPeriod := 0, Comment := '', Param1 := (Set:=0, SetMin:=0, SetMax:=0,Comment:=''), Param2 := (Set:=0, SetMin:=0, SetMax:=0,Comment:='') ),
( sName := 'a_bOperB20PitchNormalShutdownCmd', sClearName := 'Cleared', sID := '1051', a := FALSE, b := FALSE, iGroup :=1, iSetDelay :=0, iResetDelay := 0, eResetMode := MANU, eBrakeProgram := B20, eAlarmProgram := 0, Enable := TRUE, iRepetitionNumber := 0 , iRepetitionPeriod := 0, Comment := '', Param1 := (Set:=0, SetMin:=0, SetMax:=0,Comment:=''), Param2 := (Set:=0, SetMin:=0, SetMax:=0,Comment:='') ),
( sName := 'a_bHydraulicsLoadMzRam1HiWarning', sClearName := 'Hydraulic Load Hi Warning', sID := '1045', a := FALSE, b := FALSE, iGroup :=1, iSetDelay :=0, iResetDelay := 0, eResetMode := MANU, eBrakeProgram := B99, eAlarmProgram := 0, Enable := TRUE, iRepetitionNumber := 0 , iRepetitionPeriod := 0, Comment := 'Hydraulic Load Hi Warning', Param1 := (Set:=100, SetMin:=1, SetMax:=120,Comment:='kN'), Param2 := (Set:=1000, SetMin:=1, SetMax:=600000,Comment:='Nm') ),
( sName := 'a_bHydraulicsLoadMzRam1HiHiAlarm', sClearName := 'Hydraulic Load Hi Alarm', sID := '1046', a := FALSE, b := FALSE, iGroup :=1, iSetDelay :=0, iResetDelay := 0, eResetMode := MANU, eBrakeProgram := B1, eAlarmProgram := 0, Enable := TRUE, iRepetitionNumber := 0 , iRepetitionPeriod := 0, Comment := 'Hydraulic Load Hi Alarm', Param1 := (Set:=120, SetMin:=1, SetMax:=120,Comment:='kN'), Param2 := (Set:=1000, SetMin:=1, SetMax:=600000,Comment:='Nm') ),
( sName := 'a_bHydraulicsLoadMyRam2HiWarning', sClearName := 'Hydraulic Load Hi Warning', sID := '1047', a := FALSE, b := FALSE, iGroup :=1, iSetDelay :=0, iResetDelay := 0, eResetMode := MANU, eBrakeProgram := B99, eAlarmProgram := 0, Enable := TRUE, iRepetitionNumber := 0 , iRepetitionPeriod := 0, Comment := 'Hydraulic Load Hi Warning', Param1 := (Set:=490, SetMin:=1, SetMax:=500,Comment:='Kn'), Param2 := (Set:=1000, SetMin:=1, SetMax:=600000,Comment:='Nm') ),
( sName := 'a_bHydraulicsLoadMyRam2HiHiAlarm', sClearName := 'Hydraulic Load Hi Alarm', sID := '1048', a := FALSE, b := FALSE, iGroup :=1, iSetDelay :=0, iResetDelay := 0, eResetMode := MANU, eBrakeProgram := B1, eAlarmProgram := 0, Enable := TRUE, iRepetitionNumber := 0 , iRepetitionPeriod := 0, Comment := 'Hydraulic Load Hi Alarm', Param1 := (Set:=500, SetMin:=1, SetMax:=500,Comment:='Kn'), Param2 := (Set:=1000, SetMin:=1, SetMax:=600000,Comment:='Nm') ),
( sName := 'a_bHydraulicsLoadTrackingMzRAM1Warning', sClearName := 'Hydraulic Load Control Tracking Warning', sID := '1049', a := FALSE, b := FALSE, iGroup :=1, iSetDelay :=10, iResetDelay := 10, eResetMode := MANU, eBrakeProgram := B99, eAlarmProgram := 0, Enable := TRUE, iRepetitionNumber := 0 , iRepetitionPeriod := 0, Comment := 'Hydraulic Load Control Tracking Warning', Param1 := (Set:=5, SetMin:=0, SetMax:=100,Comment:=''), Param2 := (Set:=2, SetMin:=0, SetMax:=100,Comment:='') ),
( sName := 'a_bHydraulicsLoadTrackingMzRAM1Alarm', sClearName := 'Hydraulic Load Control Tracking Alarm', sID := '1050', a := FALSE, b := FALSE, iGroup :=1, iSetDelay :=10, iResetDelay := 10, eResetMode := MANU, eBrakeProgram := B20, eAlarmProgram := 0, Enable := TRUE, iRepetitionNumber := 0 , iRepetitionPeriod := 0, Comment := 'Hydraulic Load Control Tracking Alarm', Param1 := (Set:=10, SetMin:=0, SetMax:=100,Comment:=''), Param2 := (Set:=5, SetMin:=0, SetMax:=100,Comment:='') ),
( sName := 'a_bHydraulicsLoadTrackingMyRAM2Warning', sClearName := 'Hydraulic Load Control Tracking Warning', sID := '1051', a := FALSE, b := FALSE, iGroup :=1, iSetDelay :=10, iResetDelay := 10, eResetMode := MANU, eBrakeProgram := B99, eAlarmProgram := 0, Enable := TRUE, iRepetitionNumber := 0 , iRepetitionPeriod := 0, Comment := 'Hydraulic Load Control Tracking Warning', Param1 := (Set:=5, SetMin:=0, SetMax:=100,Comment:=''), Param2 := (Set:=2, SetMin:=0, SetMax:=100,Comment:='') ),
( sName := 'a_bHydraulicsLoadTrackingMyRAM2Alarm', sClearName := 'Hydraulic Load Control Tracking Alarm', sID := '1052', a := FALSE, b := FALSE, iGroup :=1, iSetDelay :=10, iResetDelay := 10, eResetMode := MANU, eBrakeProgram := B20, eAlarmProgram := 0, Enable := TRUE, iRepetitionNumber := 0 , iRepetitionPeriod := 0, Comment := 'Hydraulic Load Control Tracking Alarm', Param1 := (Set:=10, SetMin:=0, SetMax:=100,Comment:=''), Param2 := (Set:=5, SetMin:=0, SetMax:=100,Comment:='') ),
( sName := 'a_bHydraulicsLVDTSensor1Failure', sClearName := 'Hydraulics LVDT Sensor1 Failure', sID := '1053', a := FALSE, b := FALSE, iGroup :=1, iSetDelay :=0, iResetDelay := 10, eResetMode := MANU, eBrakeProgram := B99, eAlarmProgram := 0, Enable := TRUE, iRepetitionNumber := 0 , iRepetitionPeriod := 0, Comment := 'Hydraulics LVDT Sensor1 Failure', Param1 := (Set:=0, SetMin:=0, SetMax:=0,Comment:=''), Param2 := (Set:=0, SetMin:=0, SetMax:=0,Comment:='') ),
( sName := 'a_bHydraulicsLVDTSensor2Failure', sClearName := 'Hydraulics LVDT Sensor2 Failure', sID := '1054', a := FALSE, b := FALSE, iGroup :=1, iSetDelay :=0, iResetDelay := 10, eResetMode := MANU, eBrakeProgram := B99, eAlarmProgram := 0, Enable := TRUE, iRepetitionNumber := 0 , iRepetitionPeriod := 0, Comment := 'Hydraulics LVDT Sensor2 Failure', Param1 := (Set:=0, SetMin:=0, SetMax:=0,Comment:=''), Param2 := (Set:=0, SetMin:=0, SetMax:=0,Comment:='') ),
( sName := 'a_bHydraulicsLVDTSensor3Failure', sClearName := 'Hydraulics LVDT Sensor3 Failure', sID := '1055', a := FALSE, b := FALSE, iGroup :=1, iSetDelay :=0, iResetDelay := 10, eResetMode := MANU, eBrakeProgram := B99, eAlarmProgram := 0, Enable := TRUE, iRepetitionNumber := 0 , iRepetitionPeriod := 0, Comment := 'Hydraulics LVDT Sensor3 Failure', Param1 := (Set:=0, SetMin:=0, SetMax:=0,Comment:=''), Param2 := (Set:=0, SetMin:=0, SetMax:=0,Comment:='') ),
( sName := 'a_bHydraulicsLVDTSensor4Failure', sClearName := 'Hydraulics LVDT Sensor4 Failure', sID := '1056', a := FALSE, b := FALSE, iGroup :=1, iSetDelay :=0, iResetDelay := 10, eResetMode := MANU, eBrakeProgram := B99, eAlarmProgram := 0, Enable := TRUE, iRepetitionNumber := 0 , iRepetitionPeriod := 0, Comment := 'Hydraulics LVDT Sensor4 Failure', Param1 := (Set:=0, SetMin:=0, SetMax:=0,Comment:=''), Param2 := (Set:=0, SetMin:=0, SetMax:=0,Comment:='') ),
( sName := 'a_bHydraulicsLVDTSensor5Failure', sClearName := 'Hydraulics LVDT Sensor5 Failure', sID := '1057', a := FALSE, b := FALSE, iGroup :=1, iSetDelay :=0, iResetDelay := 10, eResetMode := MANU, eBrakeProgram := B99, eAlarmProgram := 0, Enable := TRUE, iRepetitionNumber := 0 , iRepetitionPeriod := 0, Comment := 'Hydraulics LVDT Sensor5 Failure', Param1 := (Set:=0, SetMin:=0, SetMax:=0,Comment:=''), Param2 := (Set:=0, SetMin:=0, SetMax:=0,Comment:='') ),
( sName := 'a_bHydraulicsLVDTSensor6Failure', sClearName := 'Hydraulics LVDT Sensor6 Failure', sID := '1058', a := FALSE, b := FALSE, iGroup :=1, iSetDelay :=0, iResetDelay := 10, eResetMode := MANU, eBrakeProgram := B99, eAlarmProgram := 0, Enable := TRUE, iRepetitionNumber := 0 , iRepetitionPeriod := 0, Comment := 'Hydraulics LVDT Sensor6 Failure', Param1 := (Set:=0, SetMin:=0, SetMax:=0,Comment:=''), Param2 := (Set:=0, SetMin:=0, SetMax:=0,Comment:='') ),
( sName := 'a_bHydraulicsLVDTSensor7Failure', sClearName := 'Hydraulics LVDT Sensor7 Failure', sID := '1059', a := FALSE, b := FALSE, iGroup :=1, iSetDelay :=0, iResetDelay := 10, eResetMode := MANU, eBrakeProgram := B99, eAlarmProgram := 0, Enable := TRUE, iRepetitionNumber := 0 , iRepetitionPeriod := 0, Comment := 'Hydraulics LVDT Sensor7 Failure', Param1 := (Set:=0, SetMin:=0, SetMax:=0,Comment:=''), Param2 := (Set:=0, SetMin:=0, SetMax:=0,Comment:='') ),
( sName := 'a_bHydraulicsLVDTSensor8Failure', sClearName := 'Hydraulics LVDT Sensor8 Failure', sID := '1060', a := FALSE, b := FALSE, iGroup :=1, iSetDelay :=0, iResetDelay := 10, eResetMode := MANU, eBrakeProgram := B99, eAlarmProgram := 0, Enable := TRUE, iRepetitionNumber := 0 , iRepetitionPeriod := 0, Comment := 'Hydraulics LVDT Sensor8 Failure', Param1 := (Set:=0, SetMin:=0, SetMax:=0,Comment:=''), Param2 := (Set:=0, SetMin:=0, SetMax:=0,Comment:='') ),
( sName := 'a_bHydraulicsMzStrainGaugeFailure', sClearName := 'Hydraulics Mz Strain Gauge Failure', sID := '1061', a := FALSE, b := FALSE, iGroup :=1, iSetDelay :=0, iResetDelay := 10, eResetMode := MANU, eBrakeProgram := B20, eAlarmProgram := 0, Enable := TRUE, iRepetitionNumber := 0 , iRepetitionPeriod := 0, Comment := 'a_bHydraulicsMzStrainGaugeFailure', Param1 := (Set:=0, SetMin:=0, SetMax:=0,Comment:=''), Param2 := (Set:=0, SetMin:=0, SetMax:=0,Comment:='') ),
( sName := 'a_bHydraulicsMyStrainGaugeFailure', sClearName := 'Hydraulics My Strain Gauge Failure', sID := '1062', a := FALSE, b := FALSE, iGroup :=1, iSetDelay :=0, iResetDelay := 10, eResetMode := MANU, eBrakeProgram := B20, eAlarmProgram := 0, Enable := TRUE, iRepetitionNumber := 0 , iRepetitionPeriod := 0, Comment := 'a_bHydraulicsMyStrainGaugeFailure', Param1 := (Set:=0, SetMin:=0, SetMax:=0,Comment:=''), Param2 := (Set:=0, SetMin:=0, SetMax:=0,Comment:='') ),
( sName := 'a_bSafetyCommsLossToSSB', sClearName := '', sID := '2001', a := FALSE, b := FALSE, iGroup :=2, iSetDelay :=0, iResetDelay := 0, eResetMode := MANU, eBrakeProgram := B4, eAlarmProgram := 0, Enable := TRUE, iRepetitionNumber := 0 , iRepetitionPeriod := 0, Comment := '', Param1 := (Set:=0, SetMin:=0, SetMax:=0,Comment:=''), Param2 := (Set:=0, SetMin:=0, SetMax:=0,Comment:='') ),
( sName := 'a_bSafetyEPO_Main_Panel', sClearName := '', sID := '2002', a := FALSE, b := FALSE, iGroup :=2, iSetDelay :=0, iResetDelay := 0, eResetMode := MANU, eBrakeProgram := B1, eAlarmProgram := 0, Enable := TRUE, iRepetitionNumber := 0 , iRepetitionPeriod := 0, Comment := '', Param1 := (Set:=0, SetMin:=0, SetMax:=0,Comment:=''), Param2 := (Set:=0, SetMin:=0, SetMax:=0,Comment:='') ),
( sName := 'a_bSafetyEPO_REMOTE', sClearName := '', sID := '2003', a := FALSE, b := FALSE, iGroup :=2, iSetDelay :=0, iResetDelay := 0, eResetMode := MANU, eBrakeProgram := B1, eAlarmProgram := 0, Enable := TRUE, iRepetitionNumber := 0 , iRepetitionPeriod := 0, Comment := '', Param1 := (Set:=0, SetMin:=0, SetMax:=0,Comment:=''), Param2 := (Set:=0, SetMin:=0, SetMax:=0,Comment:='') ),
( sName := 'a_bSafetyEPO_SCADA', sClearName := '', sID := '2004', a := FALSE, b := FALSE, iGroup :=2, iSetDelay :=0, iResetDelay := 0, eResetMode := MANU, eBrakeProgram := B1, eAlarmProgram := 0, Enable := TRUE, iRepetitionNumber := 0 , iRepetitionPeriod := 0, Comment := '', Param1 := (Set:=0, SetMin:=0, SetMax:=0,Comment:=''), Param2 := (Set:=0, SetMin:=0, SetMax:=0,Comment:='') ),
( sName := 'a_bSafetyEPO_TCP', sClearName := '', sID := '2005', a := FALSE, b := FALSE, iGroup :=2, iSetDelay :=0, iResetDelay := 0, eResetMode := MANU, eBrakeProgram := B1, eAlarmProgram := 0, Enable := TRUE, iRepetitionNumber := 0 , iRepetitionPeriod := 0, Comment := '', Param1 := (Set:=0, SetMin:=0, SetMax:=0,Comment:=''), Param2 := (Set:=0, SetMin:=0, SetMax:=0,Comment:='') ),
( sName := 'a_bSafetyOperatorRequestB1', sClearName := '', sID := '2006', a := FALSE, b := FALSE, iGroup :=2, iSetDelay :=0, iResetDelay := 0, eResetMode := MANU, eBrakeProgram := B1, eAlarmProgram := 0, Enable := TRUE, iRepetitionNumber := 0 , iRepetitionPeriod := 0, Comment := '', Param1 := (Set:=0, SetMin:=0, SetMax:=0,Comment:=''), Param2 := (Set:=0, SetMin:=0, SetMax:=0,Comment:='') ),
( sName := 'a_bSafetyOperatorRequestB4', sClearName := '', sID := '2007', a := FALSE, b := FALSE, iGroup :=2, iSetDelay :=0, iResetDelay := 0, eResetMode := MANU, eBrakeProgram := B4, eAlarmProgram := 0, Enable := TRUE, iRepetitionNumber := 0 , iRepetitionPeriod := 0, Comment := '', Param1 := (Set:=0, SetMin:=0, SetMax:=0,Comment:=''), Param2 := (Set:=0, SetMin:=0, SetMax:=0,Comment:='') ),
( sName := 'a_bSafetyOperatorRequestB9', sClearName := '', sID := '2008', a := FALSE, b := FALSE, iGroup :=2, iSetDelay :=0, iResetDelay := 0, eResetMode := MANU, eBrakeProgram := B9, eAlarmProgram := 0, Enable := TRUE, iRepetitionNumber := 0 , iRepetitionPeriod := 0, Comment := '', Param1 := (Set:=0, SetMin:=0, SetMax:=0,Comment:=''), Param2 := (Set:=0, SetMin:=0, SetMax:=0,Comment:='') ),
( sName := 'a_bSafetyEncoderPositionNOTValid', sClearName := '', sID := '2009', a := FALSE, b := FALSE, iGroup :=2, iSetDelay :=0, iResetDelay := 0, eResetMode := MANU, eBrakeProgram := B1, eAlarmProgram := 0, Enable := TRUE, iRepetitionNumber := 0 , iRepetitionPeriod := 0, Comment := '', Param1 := (Set:=0, SetMin:=0, SetMax:=0,Comment:=''), Param2 := (Set:=0, SetMin:=0, SetMax:=0,Comment:='') ),
( sName := 'a_bSafetyEncoderGroupError', sClearName := '', sID := '2010', a := FALSE, b := FALSE, iGroup :=2, iSetDelay :=0, iResetDelay := 0, eResetMode := MANU, eBrakeProgram := B1, eAlarmProgram := 0, Enable := TRUE, iRepetitionNumber := 0 , iRepetitionPeriod := 0, Comment := '', Param1 := (Set:=0, SetMin:=0, SetMax:=0,Comment:=''), Param2 := (Set:=0, SetMin:=0, SetMax:=0,Comment:='') ),
( sName := 'a_bSafetyIOGroupError', sClearName := '', sID := '2011', a := FALSE, b := FALSE, iGroup :=2, iSetDelay :=0, iResetDelay := 0, eResetMode := MANU, eBrakeProgram := B1, eAlarmProgram := 0, Enable := TRUE, iRepetitionNumber := 0 , iRepetitionPeriod := 0, Comment := '', Param1 := (Set:=0, SetMin:=0, SetMax:=0,Comment:=''), Param2 := (Set:=0, SetMin:=0, SetMax:=0,Comment:='') ),
( sName := 'a_bSafetyAngInGroupError', sClearName := '', sID := '2012', a := FALSE, b := FALSE, iGroup :=2, iSetDelay :=0, iResetDelay := 0, eResetMode := MANU, eBrakeProgram := B1, eAlarmProgram := 0, Enable := TRUE, iRepetitionNumber := 0 , iRepetitionPeriod := 0, Comment := '', Param1 := (Set:=0, SetMin:=0, SetMax:=0,Comment:=''), Param2 := (Set:=0, SetMin:=0, SetMax:=0,Comment:='') ),
( sName := 'a_bSafetyPresetGroupError', sClearName := '', sID := '2013', a := FALSE, b := FALSE, iGroup :=2, iSetDelay :=0, iResetDelay := 0, eResetMode := MANU, eBrakeProgram := B1, eAlarmProgram := 0, Enable := TRUE, iRepetitionNumber := 0 , iRepetitionPeriod := 0, Comment := '', Param1 := (Set:=0, SetMin:=0, SetMax:=0,Comment:=''), Param2 := (Set:=0, SetMin:=0, SetMax:=0,Comment:='') ),
( sName := 'a_bSafetySLS_GroupError', sClearName := '', sID := '2014', a := FALSE, b := FALSE, iGroup :=2, iSetDelay :=0, iResetDelay := 0, eResetMode := MANU, eBrakeProgram := B1, eAlarmProgram := 0, Enable := TRUE, iRepetitionNumber := 0 , iRepetitionPeriod := 0, Comment := '', Param1 := (Set:=0, SetMin:=0, SetMax:=0,Comment:=''), Param2 := (Set:=0, SetMin:=0, SetMax:=0,Comment:='') ),
( sName := 'a_bSafetyX10_PNOZ_GroupError', sClearName := '', sID := '2015', a := FALSE, b := FALSE, iGroup :=2, iSetDelay :=0, iResetDelay := 0, eResetMode := MANU, eBrakeProgram := B1, eAlarmProgram := 0, Enable := TRUE, iRepetitionNumber := 0 , iRepetitionPeriod := 0, Comment := '', Param1 := (Set:=0, SetMin:=0, SetMax:=0,Comment:=''), Param2 := (Set:=0, SetMin:=0, SetMax:=0,Comment:='') ),
( sName := 'a_bSafetyX6_ExtremFine_GroupError', sClearName := '', sID := '2016', a := FALSE, b := FALSE, iGroup :=2, iSetDelay :=0, iResetDelay := 0, eResetMode := MANU, eBrakeProgram := B1, eAlarmProgram := 0, Enable := TRUE, iRepetitionNumber := 0 , iRepetitionPeriod := 0, Comment := '', Param1 := (Set:=0, SetMin:=0, SetMax:=0,Comment:=''), Param2 := (Set:=0, SetMin:=0, SetMax:=0,Comment:='') ),
( sName := 'a_bSafetyX5_EFC_GroupError', sClearName := '', sID := '2017', a := FALSE, b := FALSE, iGroup :=2, iSetDelay :=0, iResetDelay := 0, eResetMode := MANU, eBrakeProgram := B1, eAlarmProgram := 0, Enable := TRUE, iRepetitionNumber := 0 , iRepetitionPeriod := 0, Comment := '', Param1 := (Set:=0, SetMin:=0, SetMax:=0,Comment:=''), Param2 := (Set:=0, SetMin:=0, SetMax:=0,Comment:='') ),
( sName := 'a_bSafetyFBError', sClearName := '', sID := '2018', a := FALSE, b := FALSE, iGroup :=2, iSetDelay :=0, iResetDelay := 0, eResetMode := MANU, eBrakeProgram := B1, eAlarmProgram := 0, Enable := TRUE, iRepetitionNumber := 0 , iRepetitionPeriod := 0, Comment := '', Param1 := (Set:=0, SetMin:=0, SetMax:=0,Comment:=''), Param2 := (Set:=0, SetMin:=0, SetMax:=0,Comment:='') ),
( sName := 'a_bSafetyCommError', sClearName := '', sID := '2019', a := FALSE, b := FALSE, iGroup :=2, iSetDelay :=0, iResetDelay := 0, eResetMode := MANU, eBrakeProgram := B1, eAlarmProgram := 0, Enable := TRUE, iRepetitionNumber := 0 , iRepetitionPeriod := 0, Comment := '', Param1 := (Set:=0, SetMin:=0, SetMax:=0,Comment:=''), Param2 := (Set:=0, SetMin:=0, SetMax:=0,Comment:='') ),
( sName := 'a_bSafetyOutError', sClearName := '', sID := '2020', a := FALSE, b := FALSE, iGroup :=2, iSetDelay :=0, iResetDelay := 0, eResetMode := MANU, eBrakeProgram := B1, eAlarmProgram := 0, Enable := TRUE, iRepetitionNumber := 0 , iRepetitionPeriod := 0, Comment := '', Param1 := (Set:=0, SetMin:=0, SetMax:=0,Comment:=''), Param2 := (Set:=0, SetMin:=0, SetMax:=0,Comment:='') ),
( sName := 'a_bSafetyOperatorPushButtonEstopTrip', sClearName := '', sID := '2021', a := FALSE, b := FALSE, iGroup :=2, iSetDelay :=0, iResetDelay := 0, eResetMode := MANU, eBrakeProgram := B1, eAlarmProgram := 0, Enable := TRUE, iRepetitionNumber := 0 , iRepetitionPeriod := 0, Comment := '', Param1 := (Set:=0, SetMin:=0, SetMax:=0,Comment:=''), Param2 := (Set:=0, SetMin:=0, SetMax:=0,Comment:='') ),
( sName := 'a_bSafetyHydairSystemEstopTrip', sClearName := '', sID := '2022', a := FALSE, b := FALSE, iGroup :=2, iSetDelay :=0, iResetDelay := 0, eResetMode := MANU, eBrakeProgram := B99, eAlarmProgram := 0, Enable := TRUE, iRepetitionNumber := 0 , iRepetitionPeriod := 0, Comment := '', Param1 := (Set:=0, SetMin:=0, SetMax:=0,Comment:=''), Param2 := (Set:=0, SetMin:=0, SetMax:=0,Comment:='') ),
( sName := 'a_bSafetyPTCSActivatedEstopTrip_ComssLossHydair', sClearName := '', sID := '2023', a := FALSE, b := FALSE, iGroup :=2, iSetDelay :=0, iResetDelay := 0, eResetMode := MANU, eBrakeProgram := B1, eAlarmProgram := 0, Enable := TRUE, iRepetitionNumber := 0 , iRepetitionPeriod := 0, Comment := '', Param1 := (Set:=0, SetMin:=0, SetMax:=0,Comment:=''), Param2 := (Set:=0, SetMin:=0, SetMax:=0,Comment:='') ),
( sName := 'a_bSafetyPTCSActivatedEstopTrip_ExcessiveLoadTestRig', sClearName := '', sID := '2024', a := FALSE, b := FALSE, iGroup :=2, iSetDelay :=0, iResetDelay := 0, eResetMode := MANU, eBrakeProgram := B1, eAlarmProgram := 0, Enable := TRUE, iRepetitionNumber := 0 , iRepetitionPeriod := 0, Comment := '', Param1 := (Set:=0, SetMin:=0, SetMax:=0,Comment:=''), Param2 := (Set:=0, SetMin:=0, SetMax:=0,Comment:='') ),
( sName := 'a_bSafetyPitchSystemEFCActivated', sClearName := '', sID := '2025', a := FALSE, b := FALSE, iGroup :=2, iSetDelay :=0, iResetDelay := 0, eResetMode := MANU, eBrakeProgram := B99, eAlarmProgram := 0, Enable := TRUE, iRepetitionNumber := 0 , iRepetitionPeriod := 0, Comment := '', Param1 := (Set:=0, SetMin:=0, SetMax:=0,Comment:=''), Param2 := (Set:=0, SetMin:=0, SetMax:=0,Comment:='') ),
( sName := 'a_bSafetyEstopResetReq', sClearName := '', sID := '2026', a := FALSE, b := FALSE, iGroup :=2, iSetDelay :=0, iResetDelay := 0, eResetMode := MANU, eBrakeProgram := B99, eAlarmProgram := 0, Enable := TRUE, iRepetitionNumber := 0 , iRepetitionPeriod := 0, Comment := '', Param1 := (Set:=0, SetMin:=0, SetMax:=0,Comment:=''), Param2 := (Set:=0, SetMin:=0, SetMax:=0,Comment:='') ),
( sName := 'a_bSafetyEFCResetReq', sClearName := '', sID := '2027', a := FALSE, b := FALSE, iGroup :=2, iSetDelay :=0, iResetDelay := 0, eResetMode := MANU, eBrakeProgram := B99, eAlarmProgram := 0, Enable := TRUE, iRepetitionNumber := 0 , iRepetitionPeriod := 0, Comment := '', Param1 := (Set:=0, SetMin:=0, SetMax:=0,Comment:=''), Param2 := (Set:=0, SetMin:=0, SetMax:=0,Comment:='') ),
( sName := 'a_bSafetyEstopChainClosed', sClearName := '', sID := '2028', a := FALSE, b := FALSE, iGroup :=2, iSetDelay :=0, iResetDelay := 0, eResetMode := MANU, eBrakeProgram := B99, eAlarmProgram := 0, Enable := TRUE, iRepetitionNumber := 0 , iRepetitionPeriod := 0, Comment := '', Param1 := (Set:=0, SetMin:=0, SetMax:=0,Comment:=''), Param2 := (Set:=0, SetMin:=0, SetMax:=0,Comment:='') ),
( sName := 'a_bSafetyPitchEFCChainClosed', sClearName := '', sID := '2029', a := FALSE, b := FALSE, iGroup :=2, iSetDelay :=0, iResetDelay := 0, eResetMode := MANU, eBrakeProgram := B99, eAlarmProgram := 0, Enable := TRUE, iRepetitionNumber := 0 , iRepetitionPeriod := 0, Comment := '', Param1 := (Set:=0, SetMin:=0, SetMax:=0,Comment:=''), Param2 := (Set:=0, SetMin:=0, SetMax:=0,Comment:='') ),
( sName := 'a_bConverterHeartbeatFailure', sClearName := 'Heartbeat profibus', sID := '3901', a := FALSE, b := FALSE, iGroup :=3, iSetDelay :=10, iResetDelay := 0, eResetMode := MANU, eBrakeProgram := B9, eAlarmProgram := EMAIL, Enable := FALSE, iRepetitionNumber := 0 , iRepetitionPeriod := 10, Comment := 'Heartbeat failed', Param1 := (Set:=0, SetMin:=0, SetMax:=0,Comment:=''), Param2 := (Set:=0, SetMin:=0, SetMax:=0,Comment:='') ),
( sName := 'a_bSSB_NoEFCFromTC', sClearName := 'Water level below slip ring tripped low sensor', sID := '4001', a := FALSE, b := FALSE, iGroup :=4, iSetDelay :=0, iResetDelay := 0, eResetMode := MANU, eBrakeProgram := B4, eAlarmProgram := 0, Enable := TRUE, iRepetitionNumber := 0 , iRepetitionPeriod := 0, Comment := '', Param1 := (Set:=2, SetMin:=1, SetMax:=2,Comment:=''), Param2 := (Set:=0, SetMin:=0, SetMax:=0,Comment:='') ),
( sName := 'a_bSSB_bWatchDogFromPLC', sClearName := 'bWatchDogFromPLC', sID := '4002', a := FALSE, b := FALSE, iGroup :=4, iSetDelay :=0, iResetDelay := 0, eResetMode := MANU, eBrakeProgram := B4, eAlarmProgram := 0, Enable := TRUE, iRepetitionNumber := 0 , iRepetitionPeriod := 0, Comment := '', Param1 := (Set:=0, SetMin:=0, SetMax:=0,Comment:=''), Param2 := (Set:=0, SetMin:=0, SetMax:=0,Comment:='') ),
( sName := 'a_bSSB_bAllBladesAtLimit', sClearName := 'bAllBladesAtLimit', sID := '4003', a := FALSE, b := FALSE, iGroup :=4, iSetDelay :=0, iResetDelay := 0, eResetMode := MANU, eBrakeProgram := B99, eAlarmProgram := 0, Enable := TRUE, iRepetitionNumber := 0 , iRepetitionPeriod := 0, Comment := '', Param1 := (Set:=0, SetMin:=0, SetMax:=0,Comment:=''), Param2 := (Set:=0, SetMin:=0, SetMax:=0,Comment:='') ),
( sName := 'a_bSSB_bAllBladesAtFeather', sClearName := 'bAllBladesAtFeather', sID := '4004', a := FALSE, b := FALSE, iGroup :=4, iSetDelay :=0, iResetDelay := 0, eResetMode := MANU, eBrakeProgram := B99, eAlarmProgram := 0, Enable := TRUE, iRepetitionNumber := 0 , iRepetitionPeriod := 0, Comment := '', Param1 := (Set:=0, SetMin:=0, SetMax:=0,Comment:=''), Param2 := (Set:=0, SetMin:=0, SetMax:=0,Comment:='') ),
( sName := 'a_bSSB_BusOK', sClearName := 'a_bSSB_BusOK', sID := '4005', a := FALSE, b := FALSE, iGroup :=4, iSetDelay :=0, iResetDelay := 0, eResetMode := MANU, eBrakeProgram := B99, eAlarmProgram := 0, Enable := TRUE, iRepetitionNumber := 0 , iRepetitionPeriod := 0, Comment := '', Param1 := (Set:=0, SetMin:=0, SetMax:=0,Comment:=''), Param2 := (Set:=0, SetMin:=0, SetMax:=0,Comment:='') ),
( sName := 'a_bSSB_bCriticalError', sClearName := 'a_bCriticalError', sID := '4006', a := FALSE, b := FALSE, iGroup :=4, iSetDelay :=0, iResetDelay := 0, eResetMode := MANU, eBrakeProgram := B4, eAlarmProgram := 0, Enable := TRUE, iRepetitionNumber := 0 , iRepetitionPeriod := 0, Comment := '', Param1 := (Set:=0, SetMin:=0, SetMax:=0,Comment:=''), Param2 := (Set:=0, SetMin:=0, SetMax:=0,Comment:='') ),
( sName := 'a_bSSB_bFatalError', sClearName := 'a_bFatalError', sID := '4007', a := FALSE, b := FALSE, iGroup :=4, iSetDelay :=0, iResetDelay := 0, eResetMode := MANU, eBrakeProgram := B4, eAlarmProgram := 0, Enable := TRUE, iRepetitionNumber := 0 , iRepetitionPeriod := 0, Comment := '', Param1 := (Set:=0, SetMin:=0, SetMax:=0,Comment:=''), Param2 := (Set:=0, SetMin:=0, SetMax:=0,Comment:='') ),
( sName := 'a_bSSB_bReferencingFailed', sClearName := 'bReferencingFailed', sID := '4008', a := FALSE, b := FALSE, iGroup :=4, iSetDelay :=0, iResetDelay := 0, eResetMode := MANU, eBrakeProgram := B99, eAlarmProgram := 0, Enable := TRUE, iRepetitionNumber := 0 , iRepetitionPeriod := 0, Comment := '', Param1 := (Set:=0, SetMin:=0, SetMax:=0,Comment:=''), Param2 := (Set:=0, SetMin:=0, SetMax:=0,Comment:='') ),
( sName := 'a_bSSB_ExtDI1_Lube1Flt', sClearName := 'a_ExtDI1_Lube1Flt', sID := '4009', a := FALSE, b := FALSE, iGroup :=4, iSetDelay :=0, iResetDelay := 0, eResetMode := MANU, eBrakeProgram := B99, eAlarmProgram := 0, Enable := TRUE, iRepetitionNumber := 0 , iRepetitionPeriod := 0, Comment := '', Param1 := (Set:=0, SetMin:=0, SetMax:=0,Comment:=''), Param2 := (Set:=0, SetMin:=0, SetMax:=0,Comment:='') ),
( sName := 'a_bSSB_PPA_EFC1_by_Error', sClearName := 'a_PPA_EFC1_by_Error', sID := '4010', a := FALSE, b := FALSE, iGroup :=4, iSetDelay :=0, iResetDelay := 0, eResetMode := MANU, eBrakeProgram := B4, eAlarmProgram := 0, Enable := TRUE, iRepetitionNumber := 0 , iRepetitionPeriod := 0, Comment := '', Param1 := (Set:=0, SetMin:=0, SetMax:=0,Comment:=''), Param2 := (Set:=0, SetMin:=0, SetMax:=0,Comment:='') ),
( sName := 'a_bSSB_PPA_EFC1_by_bus', sClearName := 'a_PPA_EFC1_by_bus', sID := '4011', a := FALSE, b := FALSE, iGroup :=4, iSetDelay :=0, iResetDelay := 0, eResetMode := MANU, eBrakeProgram := B99, eAlarmProgram := 0, Enable := TRUE, iRepetitionNumber := 0 , iRepetitionPeriod := 0, Comment := '', Param1 := (Set:=0, SetMin:=0, SetMax:=0,Comment:=''), Param2 := (Set:=0, SetMin:=0, SetMax:=0,Comment:='') ),
( sName := 'a_bSSB_LS_active ', sClearName := 'a_PPA_EFC1_active', sID := '4012', a := FALSE, b := FALSE, iGroup :=4, iSetDelay :=0, iResetDelay := 0, eResetMode := MANU, eBrakeProgram := B99, eAlarmProgram := 0, Enable := TRUE, iRepetitionNumber := 0 , iRepetitionPeriod := 0, Comment := '', Param1 := (Set:=0, SetMin:=0, SetMax:=0,Comment:=''), Param2 := (Set:=0, SetMin:=0, SetMax:=0,Comment:='') ),
( sName := 'a_bSSB_SWLS', sClearName := 'a_bSSB_SWLS', sID := '4013', a := FALSE, b := FALSE, iGroup :=4, iSetDelay :=0, iResetDelay := 0, eResetMode := MANU, eBrakeProgram := B99, eAlarmProgram := 0, Enable := TRUE, iRepetitionNumber := 0 , iRepetitionPeriod := 0, Comment := '', Param1 := (Set:=0, SetMin:=0, SetMax:=0,Comment:=''), Param2 := (Set:=0, SetMin:=0, SetMax:=0,Comment:='') ),
( sName := 'a_bSSB_Bypass1stlimitactive', sClearName := 'a_bSSB_Bypass1stlimitactive', sID := '4014', a := FALSE, b := FALSE, iGroup :=4, iSetDelay :=0, iResetDelay := 0, eResetMode := MANU, eBrakeProgram := B99, eAlarmProgram := 0, Enable := TRUE, iRepetitionNumber := 0 , iRepetitionPeriod := 0, Comment := '', Param1 := (Set:=0, SetMin:=0, SetMax:=0,Comment:=''), Param2 := (Set:=0, SetMin:=0, SetMax:=0,Comment:='') ),
( sName := 'a_bSSB_MainsWarning', sClearName := 'Mains ok (1 = ok, 0 = general warning)', sID := '4015', a := FALSE, b := FALSE, iGroup :=4, iSetDelay :=0, iResetDelay := 0, eResetMode := MANU, eBrakeProgram := B99, eAlarmProgram := 0, Enable := TRUE, iRepetitionNumber := 0 , iRepetitionPeriod := 0, Comment := '', Param1 := (Set:=0, SetMin:=0, SetMax:=0,Comment:=''), Param2 := (Set:=0, SetMin:=0, SetMax:=0,Comment:='') ),
( sName := 'a_bSSB_CurrentBackup_heaterLow', sClearName := 'a_bSSB_CurrentBackup_heaterLow', sID := '4016', a := FALSE, b := FALSE, iGroup :=4, iSetDelay :=0, iResetDelay := 0, eResetMode := MANU, eBrakeProgram := B99, eAlarmProgram := 0, Enable := TRUE, iRepetitionNumber := 0 , iRepetitionPeriod := 0, Comment := '', Param1 := (Set:=0, SetMin:=0, SetMax:=0,Comment:=''), Param2 := (Set:=0, SetMin:=0, SetMax:=0,Comment:='') ),
( sName := 'a_bSSB_Crit_InternEncoderDeviation', sClearName := '; (motor encoder - blade encoder) > uMAX_DEVIATION', sID := '4017', a := FALSE, b := FALSE, iGroup :=4, iSetDelay :=0, iResetDelay := 0, eResetMode := MANU, eBrakeProgram := B4, eAlarmProgram := 0, Enable := TRUE, iRepetitionNumber := 0 , iRepetitionPeriod := 0, Comment := '', Param1 := (Set:=0, SetMin:=0, SetMax:=0,Comment:=''), Param2 := (Set:=0, SetMin:=0, SetMax:=0,Comment:='') ),
( sName := 'a_bSSB_Crit_ExternEncoderDeviation', sClearName := 'a_bSSB_ExternEncoderDeviation', sID := '4018', a := FALSE, b := FALSE, iGroup :=4, iSetDelay :=0, iResetDelay := 0, eResetMode := MANU, eBrakeProgram := B4, eAlarmProgram := 0, Enable := TRUE, iRepetitionNumber := 0 , iRepetitionPeriod := 0, Comment := '', Param1 := (Set:=0, SetMin:=0, SetMax:=0,Comment:=''), Param2 := (Set:=0, SetMin:=0, SetMax:=0,Comment:='') ),
( sName := 'a_bSSB_Backup_Charger_Not_Working', sClearName := '', sID := '4019', a := FALSE, b := FALSE, iGroup :=4, iSetDelay :=0, iResetDelay := 0, eResetMode := MANU, eBrakeProgram := B4, eAlarmProgram := 0, Enable := TRUE, iRepetitionNumber := 0 , iRepetitionPeriod := 0, Comment := '', Param1 := (Set:=0, SetMin:=0, SetMax:=0,Comment:=''), Param2 := (Set:=0, SetMin:=0, SetMax:=0,Comment:='') ),
( sName := 'a_bSSB_Crit_Backup_heating', sClearName := 'a_bSSB_Backup_heating', sID := '4020', a := FALSE, b := FALSE, iGroup :=4, iSetDelay :=0, iResetDelay := 0, eResetMode := MANU, eBrakeProgram := B99, eAlarmProgram := 0, Enable := TRUE, iRepetitionNumber := 0 , iRepetitionPeriod := 0, Comment := '', Param1 := (Set:=0, SetMin:=0, SetMax:=0,Comment:=''), Param2 := (Set:=0, SetMin:=0, SetMax:=0,Comment:='') ),
( sName := 'a_bSSB_Crit_Mains_Not_OK', sClearName := 'a_bSSB_Mains not OK', sID := '4021', a := FALSE, b := FALSE, iGroup :=4, iSetDelay :=0, iResetDelay := 0, eResetMode := MANU, eBrakeProgram := B4, eAlarmProgram := 0, Enable := TRUE, iRepetitionNumber := 0 , iRepetitionPeriod := 0, Comment := '', Param1 := (Set:=0, SetMin:=0, SetMax:=0,Comment:=''), Param2 := (Set:=0, SetMin:=0, SetMax:=0,Comment:='') ),
( sName := 'a_bPPA_ALM_NH', sClearName := '', sID := '4022', a := FALSE, b := FALSE, iGroup :=4, iSetDelay :=0, iResetDelay := 0, eResetMode := MANU, eBrakeProgram := B99, eAlarmProgram := 0, Enable := TRUE, iRepetitionNumber := 0 , iRepetitionPeriod := 0, Comment := 'Error Overspeed', Param1 := (Set:=0, SetMin:=0, SetMax:=0,Comment:=''), Param2 := (Set:=0, SetMin:=0, SetMax:=0,Comment:='') ),
( sName := 'a_bPPA_ALM_UP', sClearName := '', sID := '4023', a := FALSE, b := FALSE, iGroup :=4, iSetDelay :=0, iResetDelay := 0, eResetMode := MANU, eBrakeProgram := B99, eAlarmProgram := 0, Enable := TRUE, iRepetitionNumber := 0 , iRepetitionPeriod := 0, Comment := 'Error Grid(UP)', Param1 := (Set:=0, SetMin:=0, SetMax:=0,Comment:=''), Param2 := (Set:=0, SetMin:=0, SetMax:=0,Comment:='') ),
( sName := 'a_bPPA_ALM_VH', sClearName := '', sID := '4024', a := FALSE, b := FALSE, iGroup :=4, iSetDelay :=0, iResetDelay := 0, eResetMode := MANU, eBrakeProgram := B99, eAlarmProgram := 0, Enable := TRUE, iRepetitionNumber := 0 , iRepetitionPeriod := 0, Comment := 'Error DC Link High', Param1 := (Set:=0, SetMin:=0, SetMax:=0,Comment:=''), Param2 := (Set:=0, SetMin:=0, SetMax:=0,Comment:='') ),
( sName := 'a_bPPA_ALM_VL', sClearName := '', sID := '4025', a := FALSE, b := FALSE, iGroup :=4, iSetDelay :=0, iResetDelay := 0, eResetMode := MANU, eBrakeProgram := B99, eAlarmProgram := 0, Enable := TRUE, iRepetitionNumber := 0 , iRepetitionPeriod := 0, Comment := 'Error DC Link Low', Param1 := (Set:=0, SetMin:=0, SetMax:=0,Comment:=''), Param2 := (Set:=0, SetMin:=0, SetMax:=0,Comment:='') ),
( sName := 'a_bPPA_ALM_VU', sClearName := '', sID := '4026', a := FALSE, b := FALSE, iGroup :=4, iSetDelay :=0, iResetDelay := 0, eResetMode := MANU, eBrakeProgram := B99, eAlarmProgram := 0, Enable := TRUE, iRepetitionNumber := 0 , iRepetitionPeriod := 0, Comment := 'Error DC Link unplausable', Param1 := (Set:=0, SetMin:=0, SetMax:=0,Comment:=''), Param2 := (Set:=0, SetMin:=0, SetMax:=0,Comment:='') ),
( sName := 'a_bPPA_ALM_OO', sClearName := '', sID := '4027', a := FALSE, b := FALSE, iGroup :=4, iSetDelay :=0, iResetDelay := 0, eResetMode := MANU, eBrakeProgram := B99, eAlarmProgram := 0, Enable := TRUE, iRepetitionNumber := 0 , iRepetitionPeriod := 0, Comment := 'Error Open Output', Param1 := (Set:=0, SetMin:=0, SetMax:=0,Comment:=''), Param2 := (Set:=0, SetMin:=0, SetMax:=0,Comment:='') ),
( sName := 'a_bPPA_ALM_RB', sClearName := '', sID := '4028', a := FALSE, b := FALSE, iGroup :=4, iSetDelay :=0, iResetDelay := 0, eResetMode := MANU, eBrakeProgram := B99, eAlarmProgram := 0, Enable := TRUE, iRepetitionNumber := 0 , iRepetitionPeriod := 0, Comment := 'Error Brake Chopper', Param1 := (Set:=0, SetMin:=0, SetMax:=0,Comment:=''), Param2 := (Set:=0, SetMin:=0, SetMax:=0,Comment:='') ),
( sName := 'a_bPPA_ALM_OF', sClearName := '', sID := '4029', a := FALSE, b := FALSE, iGroup :=4, iSetDelay :=0, iResetDelay := 0, eResetMode := MANU, eBrakeProgram := B99, eAlarmProgram := 0, Enable := TRUE, iRepetitionNumber := 0 , iRepetitionPeriod := 0, Comment := 'Error Overload IGBT', Param1 := (Set:=0, SetMin:=0, SetMax:=0,Comment:=''), Param2 := (Set:=0, SetMin:=0, SetMax:=0,Comment:='') ),
( sName := 'a_bPPA_ALM_OC', sClearName := '', sID := '4030', a := FALSE, b := FALSE, iGroup :=4, iSetDelay :=0, iResetDelay := 0, eResetMode := MANU, eBrakeProgram := B99, eAlarmProgram := 0, Enable := TRUE, iRepetitionNumber := 0 , iRepetitionPeriod := 0, Comment := 'Error Overcurrent', Param1 := (Set:=0, SetMin:=0, SetMax:=0,Comment:=''), Param2 := (Set:=0, SetMin:=0, SetMax:=0,Comment:='') ),
( sName := 'a_bPPA_ALM_CF', sClearName := '', sID := '4031', a := FALSE, b := FALSE, iGroup :=4, iSetDelay :=0, iResetDelay := 0, eResetMode := MANU, eBrakeProgram := B99, eAlarmProgram := 0, Enable := TRUE, iRepetitionNumber := 0 , iRepetitionPeriod := 0, Comment := 'Error Current -V', Param1 := (Set:=0, SetMin:=0, SetMax:=0,Comment:=''), Param2 := (Set:=0, SetMin:=0, SetMax:=0,Comment:='') ),
( sName := 'a_bPPA_ALM_IS', sClearName := '', sID := '4032', a := FALSE, b := FALSE, iGroup :=4, iSetDelay :=0, iResetDelay := 0, eResetMode := MANU, eBrakeProgram := B99, eAlarmProgram := 0, Enable := TRUE, iRepetitionNumber := 0 , iRepetitionPeriod := 0, Comment := 'Error Internal Supply', Param1 := (Set:=0, SetMin:=0, SetMax:=0,Comment:=''), Param2 := (Set:=0, SetMin:=0, SetMax:=0,Comment:='') ),
( sName := 'a_bPPA_ALM_VE', sClearName := '', sID := '4033', a := FALSE, b := FALSE, iGroup :=4, iSetDelay :=0, iResetDelay := 0, eResetMode := MANU, eBrakeProgram := B99, eAlarmProgram := 0, Enable := TRUE, iRepetitionNumber := 0 , iRepetitionPeriod := 0, Comment := 'Error Electronic supply', Param1 := (Set:=0, SetMin:=0, SetMax:=0,Comment:=''), Param2 := (Set:=0, SetMin:=0, SetMax:=0,Comment:='') ),
( sName := 'a_bPPA_ALM_HF', sClearName := '', sID := '4034', a := FALSE, b := FALSE, iGroup :=4, iSetDelay :=0, iResetDelay := 0, eResetMode := MANU, eBrakeProgram := B99, eAlarmProgram := 0, Enable := TRUE, iRepetitionNumber := 0 , iRepetitionPeriod := 0, Comment := 'Error Hardware Failure', Param1 := (Set:=0, SetMin:=0, SetMax:=0,Comment:=''), Param2 := (Set:=0, SetMin:=0, SetMax:=0,Comment:='') ),
( sName := 'a_bPPA_ALM_PE', sClearName := '', sID := '4035', a := FALSE, b := FALSE, iGroup :=4, iSetDelay :=0, iResetDelay := 0, eResetMode := MANU, eBrakeProgram := B99, eAlarmProgram := 0, Enable := TRUE, iRepetitionNumber := 0 , iRepetitionPeriod := 0, Comment := 'Error Parameter Loading', Param1 := (Set:=0, SetMin:=0, SetMax:=0,Comment:=''), Param2 := (Set:=0, SetMin:=0, SetMax:=0,Comment:='') ),
( sName := 'a_bPPA_ALM_MM', sClearName := '', sID := '4036', a := FALSE, b := FALSE, iGroup :=4, iSetDelay :=0, iResetDelay := 0, eResetMode := MANU, eBrakeProgram := B99, eAlarmProgram := 0, Enable := TRUE, iRepetitionNumber := 0 , iRepetitionPeriod := 0, Comment := 'Error Motor lxt', Param1 := (Set:=0, SetMin:=0, SetMax:=0,Comment:=''), Param2 := (Set:=0, SetMin:=0, SetMax:=0,Comment:='') ),
( sName := 'a_bPPA_ALM_CP', sClearName := '', sID := '4037', a := FALSE, b := FALSE, iGroup :=4, iSetDelay :=0, iResetDelay := 0, eResetMode := MANU, eBrakeProgram := B99, eAlarmProgram := 0, Enable := TRUE, iRepetitionNumber := 0 , iRepetitionPeriod := 0, Comment := 'Error Preogram', Param1 := (Set:=0, SetMin:=0, SetMax:=0,Comment:=''), Param2 := (Set:=0, SetMin:=0, SetMax:=0,Comment:='') ),
( sName := 'a_bPPA_ALM_EE', sClearName := '', sID := '4038', a := FALSE, b := FALSE, iGroup :=4, iSetDelay :=0, iResetDelay := 0, eResetMode := MANU, eBrakeProgram := B99, eAlarmProgram := 0, Enable := TRUE, iRepetitionNumber := 0 , iRepetitionPeriod := 0, Comment := 'Error EEPROM', Param1 := (Set:=0, SetMin:=0, SetMax:=0,Comment:=''), Param2 := (Set:=0, SetMin:=0, SetMax:=0,Comment:='') ),
( sName := 'a_bPPA_ALM_SB', sClearName := '', sID := '4039', a := FALSE, b := FALSE, iGroup :=4, iSetDelay :=0, iResetDelay := 0, eResetMode := MANU, eBrakeProgram := B99, eAlarmProgram := 0, Enable := TRUE, iRepetitionNumber := 0 , iRepetitionPeriod := 0, Comment := 'Error SSB Bus', Param1 := (Set:=0, SetMin:=0, SetMax:=0,Comment:=''), Param2 := (Set:=0, SetMin:=0, SetMax:=0,Comment:='') ),
( sName := 'a_bPPA_ALM_E1', sClearName := '', sID := '4040', a := FALSE, b := FALSE, iGroup :=4, iSetDelay :=0, iResetDelay := 0, eResetMode := MANU, eBrakeProgram := B99, eAlarmProgram := 0, Enable := TRUE, iRepetitionNumber := 0 , iRepetitionPeriod := 0, Comment := 'Error Encoder 1', Param1 := (Set:=0, SetMin:=0, SetMax:=0,Comment:=''), Param2 := (Set:=0, SetMin:=0, SetMax:=0,Comment:='') ),
( sName := 'a_bPPA_ALM_E2', sClearName := '', sID := '4041', a := FALSE, b := FALSE, iGroup :=4, iSetDelay :=0, iResetDelay := 0, eResetMode := MANU, eBrakeProgram := B99, eAlarmProgram := 0, Enable := TRUE, iRepetitionNumber := 0 , iRepetitionPeriod := 0, Comment := 'Error Encoder 2', Param1 := (Set:=0, SetMin:=0, SetMax:=0,Comment:=''), Param2 := (Set:=0, SetMin:=0, SetMax:=0,Comment:='') ),
( sName := 'a_bPPA_ALM_SL', sClearName := '', sID := '4042', a := FALSE, b := FALSE, iGroup :=4, iSetDelay :=0, iResetDelay := 0, eResetMode := MANU, eBrakeProgram := B99, eAlarmProgram := 0, Enable := TRUE, iRepetitionNumber := 0 , iRepetitionPeriod := 0, Comment := 'Error SWLS', Param1 := (Set:=0, SetMin:=0, SetMax:=0,Comment:=''), Param2 := (Set:=0, SetMin:=0, SetMax:=0,Comment:='') ),
( sName := 'a_bPPA_ALM_SF', sClearName := '', sID := '4043', a := FALSE, b := FALSE, iGroup :=4, iSetDelay :=0, iResetDelay := 0, eResetMode := MANU, eBrakeProgram := B99, eAlarmProgram := 0, Enable := TRUE, iRepetitionNumber := 0 , iRepetitionPeriod := 0, Comment := 'Error Speed Feedback', Param1 := (Set:=0, SetMin:=0, SetMax:=0,Comment:=''), Param2 := (Set:=0, SetMin:=0, SetMax:=0,Comment:='') ),
( sName := 'a_bPPA_ALM_PF', sClearName := '', sID := '4044', a := FALSE, b := FALSE, iGroup :=4, iSetDelay :=0, iResetDelay := 0, eResetMode := MANU, eBrakeProgram := B99, eAlarmProgram := 0, Enable := TRUE, iRepetitionNumber := 0 , iRepetitionPeriod := 0, Comment := 'Error Position', Param1 := (Set:=0, SetMin:=0, SetMax:=0,Comment:=''), Param2 := (Set:=0, SetMin:=0, SetMax:=0,Comment:='') ),
( sName := 'a_bPPA_ALM_BH', sClearName := '', sID := '4045', a := FALSE, b := FALSE, iGroup :=4, iSetDelay :=0, iResetDelay := 0, eResetMode := MANU, eBrakeProgram := B99, eAlarmProgram := 0, Enable := TRUE, iRepetitionNumber := 0 , iRepetitionPeriod := 0, Comment := 'Error Brake Current High', Param1 := (Set:=0, SetMin:=0, SetMax:=0,Comment:=''), Param2 := (Set:=0, SetMin:=0, SetMax:=0,Comment:='') ),
( sName := 'a_bPPA_ALM_BL', sClearName := '', sID := '4046', a := FALSE, b := FALSE, iGroup :=4, iSetDelay :=0, iResetDelay := 0, eResetMode := MANU, eBrakeProgram := B99, eAlarmProgram := 0, Enable := TRUE, iRepetitionNumber := 0 , iRepetitionPeriod := 0, Comment := 'Error Brake Current Low', Param1 := (Set:=0, SetMin:=0, SetMax:=0,Comment:=''), Param2 := (Set:=0, SetMin:=0, SetMax:=0,Comment:='') ),
( sName := 'a_bPPA_ALM_BD', sClearName := '', sID := '4047', a := FALSE, b := FALSE, iGroup :=4, iSetDelay :=0, iResetDelay := 0, eResetMode := MANU, eBrakeProgram := B99, eAlarmProgram := 0, Enable := TRUE, iRepetitionNumber := 0 , iRepetitionPeriod := 0, Comment := 'Error Brake Drive', Param1 := (Set:=0, SetMin:=0, SetMax:=0,Comment:=''), Param2 := (Set:=0, SetMin:=0, SetMax:=0,Comment:='') ),
( sName := 'a_bPPA_ALM_MT', sClearName := '', sID := '4048', a := FALSE, b := FALSE, iGroup :=4, iSetDelay :=0, iResetDelay := 0, eResetMode := MANU, eBrakeProgram := B99, eAlarmProgram := 0, Enable := TRUE, iRepetitionNumber := 0 , iRepetitionPeriod := 0, Comment := 'Error Motor Temperature', Param1 := (Set:=0, SetMin:=0, SetMax:=0,Comment:=''), Param2 := (Set:=0, SetMin:=0, SetMax:=0,Comment:='') ),
( sName := 'a_bPPA_ALM_HT', sClearName := '', sID := '4049', a := FALSE, b := FALSE, iGroup :=4, iSetDelay :=0, iResetDelay := 0, eResetMode := MANU, eBrakeProgram := B99, eAlarmProgram := 0, Enable := TRUE, iRepetitionNumber := 0 , iRepetitionPeriod := 0, Comment := 'Error Heat Sink Temp', Param1 := (Set:=0, SetMin:=0, SetMax:=0,Comment:=''), Param2 := (Set:=0, SetMin:=0, SetMax:=0,Comment:='') ),
( sName := 'a_bPPA_ALM_TL', sClearName := '', sID := '4050', a := FALSE, b := FALSE, iGroup :=4, iSetDelay :=0, iResetDelay := 0, eResetMode := MANU, eBrakeProgram := B99, eAlarmProgram := 0, Enable := TRUE, iRepetitionNumber := 0 , iRepetitionPeriod := 0, Comment := 'Error Control board Temp Low', Param1 := (Set:=0, SetMin:=0, SetMax:=0,Comment:=''), Param2 := (Set:=0, SetMin:=0, SetMax:=0,Comment:='') ),
( sName := 'a_bPPA_ALM_T1', sClearName := '', sID := '4051', a := FALSE, b := FALSE, iGroup :=4, iSetDelay :=0, iResetDelay := 0, eResetMode := MANU, eBrakeProgram := B99, eAlarmProgram := 0, Enable := TRUE, iRepetitionNumber := 0 , iRepetitionPeriod := 0, Comment := 'Error Control board temp High', Param1 := (Set:=0, SetMin:=0, SetMax:=0,Comment:=''), Param2 := (Set:=0, SetMin:=0, SetMax:=0,Comment:='') ),
( sName := 'a_bPPA_ALM_T2', sClearName := '', sID := '4052', a := FALSE, b := FALSE, iGroup :=4, iSetDelay :=0, iResetDelay := 0, eResetMode := MANU, eBrakeProgram := B99, eAlarmProgram := 0, Enable := TRUE, iRepetitionNumber := 0 , iRepetitionPeriod := 0, Comment := 'Error Power supply temp', Param1 := (Set:=0, SetMin:=0, SetMax:=0,Comment:=''), Param2 := (Set:=0, SetMin:=0, SetMax:=0,Comment:='') ),
( sName := 'a_bPPA_ALM_CR', sClearName := '', sID := '4053', a := FALSE, b := FALSE, iGroup :=4, iSetDelay :=0, iResetDelay := 0, eResetMode := MANU, eBrakeProgram := B99, eAlarmProgram := 0, Enable := TRUE, iRepetitionNumber := 0 , iRepetitionPeriod := 0, Comment := 'Error Controlled Rectifier', Param1 := (Set:=0, SetMin:=0, SetMax:=0,Comment:=''), Param2 := (Set:=0, SetMin:=0, SetMax:=0,Comment:='') ),
( sName := 'a_bPPA_ALM_TT', sClearName := '', sID := '4054', a := FALSE, b := FALSE, iGroup :=4, iSetDelay :=0, iResetDelay := 0, eResetMode := MANU, eBrakeProgram := B99, eAlarmProgram := 0, Enable := TRUE, iRepetitionNumber := 0 , iRepetitionPeriod := 0, Comment := 'Error IGBT Temp', Param1 := (Set:=0, SetMin:=0, SetMax:=0,Comment:=''), Param2 := (Set:=0, SetMin:=0, SetMax:=0,Comment:='') ),
( sName := 'a_bPPA_ALM_S1', sClearName := '', sID := '4055', a := FALSE, b := FALSE, iGroup :=4, iSetDelay :=0, iResetDelay := 0, eResetMode := MANU, eBrakeProgram := B99, eAlarmProgram := 0, Enable := TRUE, iRepetitionNumber := 0 , iRepetitionPeriod := 0, Comment := 'Error ICO Slave 1', Param1 := (Set:=0, SetMin:=0, SetMax:=0,Comment:=''), Param2 := (Set:=0, SetMin:=0, SetMax:=0,Comment:='') ),
( sName := 'a_bPPA_ALM_S2', sClearName := '', sID := '4056', a := FALSE, b := FALSE, iGroup :=4, iSetDelay :=0, iResetDelay := 0, eResetMode := MANU, eBrakeProgram := B99, eAlarmProgram := 0, Enable := TRUE, iRepetitionNumber := 0 , iRepetitionPeriod := 0, Comment := 'Error ICO Slave 2', Param1 := (Set:=0, SetMin:=0, SetMax:=0,Comment:=''), Param2 := (Set:=0, SetMin:=0, SetMax:=0,Comment:='') ),
( sName := 'a_bPPA_ALM_HB', sClearName := '', sID := '4057', a := FALSE, b := FALSE, iGroup :=4, iSetDelay :=0, iResetDelay := 0, eResetMode := MANU, eBrakeProgram := B99, eAlarmProgram := 0, Enable := TRUE, iRepetitionNumber := 0 , iRepetitionPeriod := 0, Comment := 'Error Back up voltage high', Param1 := (Set:=0, SetMin:=0, SetMax:=0,Comment:=''), Param2 := (Set:=0, SetMin:=0, SetMax:=0,Comment:='') ),
( sName := 'a_bPPA_ALM_LB', sClearName := '', sID := '4058', a := FALSE, b := FALSE, iGroup :=4, iSetDelay :=0, iResetDelay := 0, eResetMode := MANU, eBrakeProgram := B99, eAlarmProgram := 0, Enable := TRUE, iRepetitionNumber := 0 , iRepetitionPeriod := 0, Comment := 'Error Back up voltage Low', Param1 := (Set:=0, SetMin:=0, SetMax:=0,Comment:=''), Param2 := (Set:=0, SetMin:=0, SetMax:=0,Comment:='') ),
( sName := 'a_bPPA_ALM_RS', sClearName := '', sID := '4059', a := FALSE, b := FALSE, iGroup :=4, iSetDelay :=0, iResetDelay := 0, eResetMode := MANU, eBrakeProgram := B99, eAlarmProgram := 0, Enable := TRUE, iRepetitionNumber := 0 , iRepetitionPeriod := 0, Comment := 'Error Resolver sync', Param1 := (Set:=0, SetMin:=0, SetMax:=0,Comment:=''), Param2 := (Set:=0, SetMin:=0, SetMax:=0,Comment:='') ),
( sName := 'a_bPPA_ALM_RR', sClearName := '', sID := '4060', a := FALSE, b := FALSE, iGroup :=4, iSetDelay :=0, iResetDelay := 0, eResetMode := MANU, eBrakeProgram := B99, eAlarmProgram := 0, Enable := TRUE, iRepetitionNumber := 0 , iRepetitionPeriod := 0, Comment := 'Error Resolver Reference', Param1 := (Set:=0, SetMin:=0, SetMax:=0,Comment:=''), Param2 := (Set:=0, SetMin:=0, SetMax:=0,Comment:='') ),
( sName := 'a_bPPA_ALM_CE', sClearName := '', sID := '4061', a := FALSE, b := FALSE, iGroup :=4, iSetDelay :=0, iResetDelay := 0, eResetMode := MANU, eBrakeProgram := B99, eAlarmProgram := 0, Enable := TRUE, iRepetitionNumber := 0 , iRepetitionPeriod := 0, Comment := 'Error CANext', Param1 := (Set:=0, SetMin:=0, SetMax:=0,Comment:=''), Param2 := (Set:=0, SetMin:=0, SetMax:=0,Comment:='') ),
( sName := 'a_bPPA_ALM_C2', sClearName := '', sID := '4062', a := FALSE, b := FALSE, iGroup :=4, iSetDelay :=0, iResetDelay := 0, eResetMode := MANU, eBrakeProgram := B99, eAlarmProgram := 0, Enable := TRUE, iRepetitionNumber := 0 , iRepetitionPeriod := 0, Comment := 'Error ', Param1 := (Set:=0, SetMin:=0, SetMax:=0,Comment:=''), Param2 := (Set:=0, SetMin:=0, SetMax:=0,Comment:='') ),
( sName := 'a_bPPA_ALM_PS', sClearName := '', sID := '4063', a := FALSE, b := FALSE, iGroup :=4, iSetDelay :=0, iResetDelay := 0, eResetMode := MANU, eBrakeProgram := B99, eAlarmProgram := 0, Enable := TRUE, iRepetitionNumber := 0 , iRepetitionPeriod := 0, Comment := 'Error ', Param1 := (Set:=0, SetMin:=0, SetMax:=0,Comment:=''), Param2 := (Set:=0, SetMin:=0, SetMax:=0,Comment:='') ),
( sName := 'a_bPPA_ALM_QC', sClearName := '', sID := '4064', a := FALSE, b := FALSE, iGroup :=4, iSetDelay :=0, iResetDelay := 0, eResetMode := MANU, eBrakeProgram := B99, eAlarmProgram := 0, Enable := TRUE, iRepetitionNumber := 0 , iRepetitionPeriod := 0, Comment := 'Error ', Param1 := (Set:=0, SetMin:=0, SetMax:=0,Comment:=''), Param2 := (Set:=0, SetMin:=0, SetMax:=0,Comment:='') ),
( sName := 'a_bPPA_ALM_RE', sClearName := '', sID := '4065', a := FALSE, b := FALSE, iGroup :=4, iSetDelay :=0, iResetDelay := 0, eResetMode := MANU, eBrakeProgram := B99, eAlarmProgram := 0, Enable := TRUE, iRepetitionNumber := 0 , iRepetitionPeriod := 0, Comment := 'Error Value Range Extended', Param1 := (Set:=0, SetMin:=0, SetMax:=0,Comment:=''), Param2 := (Set:=0, SetMin:=0, SetMax:=0,Comment:='') ),
( sName := 'a_bNoSSBBusFailureANDAllSlavesStatusOnline', sClearName := '', sID := '4066', a := FALSE, b := FALSE, iGroup :=4, iSetDelay :=0, iResetDelay := 0, eResetMode := MANU, eBrakeProgram := B99, eAlarmProgram := 0, Enable := TRUE, iRepetitionNumber := 0 , iRepetitionPeriod := 0, Comment := '', Param1 := (Set:=0, SetMin:=0, SetMax:=0,Comment:=''), Param2 := (Set:=0, SetMin:=0, SetMax:=0,Comment:='') ),
( sName := 'a_bNoCommunicationTOANYSlave', sClearName := '', sID := '4067', a := FALSE, b := FALSE, iGroup :=4, iSetDelay :=0, iResetDelay := 0, eResetMode := MANU, eBrakeProgram := B99, eAlarmProgram := 0, Enable := TRUE, iRepetitionNumber := 0 , iRepetitionPeriod := 0, Comment := 'System Fatal Error bit 4 SSB to any slave not ok', Param1 := (Set:=0, SetMin:=0, SetMax:=0,Comment:=''), Param2 := (Set:=0, SetMin:=0, SetMax:=0,Comment:='') ),
( sName := 'a_bNoCommunicationTOPLCMaster', sClearName := '', sID := '4068', a := FALSE, b := FALSE, iGroup :=4, iSetDelay :=0, iResetDelay := 0, eResetMode := MANU, eBrakeProgram := B99, eAlarmProgram := 0, Enable := TRUE, iRepetitionNumber := 0 , iRepetitionPeriod := 0, Comment := '', Param1 := (Set:=0, SetMin:=0, SetMax:=0,Comment:=''), Param2 := (Set:=0, SetMin:=0, SetMax:=0,Comment:='') ),
( sName := 'a_bNoCommunicationTOSlave1_SCI', sClearName := '', sID := '4069', a := FALSE, b := FALSE, iGroup :=4, iSetDelay :=0, iResetDelay := 0, eResetMode := MANU, eBrakeProgram := B99, eAlarmProgram := 0, Enable := TRUE, iRepetitionNumber := 0 , iRepetitionPeriod := 0, Comment := '', Param1 := (Set:=0, SetMin:=0, SetMax:=0,Comment:=''), Param2 := (Set:=0, SetMin:=0, SetMax:=0,Comment:='') ),
( sName := 'a_bNoCommunicationTOSlave2_PPAM1', sClearName := '', sID := '4070', a := FALSE, b := FALSE, iGroup :=4, iSetDelay :=0, iResetDelay := 0, eResetMode := MANU, eBrakeProgram := B99, eAlarmProgram := 0, Enable := TRUE, iRepetitionNumber := 0 , iRepetitionPeriod := 0, Comment := '', Param1 := (Set:=0, SetMin:=0, SetMax:=0,Comment:=''), Param2 := (Set:=0, SetMin:=0, SetMax:=0,Comment:='') ),
( sName := 'a_bNoCommunicationTOSlave3_PPAM2', sClearName := '', sID := '4071', a := FALSE, b := FALSE, iGroup :=4, iSetDelay :=0, iResetDelay := 0, eResetMode := MANU, eBrakeProgram := B99, eAlarmProgram := 0, Enable := TRUE, iRepetitionNumber := 0 , iRepetitionPeriod := 0, Comment := '', Param1 := (Set:=0, SetMin:=0, SetMax:=0,Comment:=''), Param2 := (Set:=0, SetMin:=0, SetMax:=0,Comment:='') ),
( sName := 'a_bNoCommunicationTOSlave4_PPAM3', sClearName := '', sID := '4072', a := FALSE, b := FALSE, iGroup :=4, iSetDelay :=0, iResetDelay := 0, eResetMode := MANU, eBrakeProgram := B99, eAlarmProgram := 0, Enable := TRUE, iRepetitionNumber := 0 , iRepetitionPeriod := 0, Comment := '', Param1 := (Set:=0, SetMin:=0, SetMax:=0,Comment:=''), Param2 := (Set:=0, SetMin:=0, SetMax:=0,Comment:='') ),
( sName := 'a_bNoCommunicationToPLCFromSlave2PPAMaster1', sClearName := '', sID := '4073', a := FALSE, b := FALSE, iGroup :=4, iSetDelay :=0, iResetDelay := 0, eResetMode := MANU, eBrakeProgram := B99, eAlarmProgram := 0, Enable := TRUE, iRepetitionNumber := 0 , iRepetitionPeriod := 0, Comment := 'system fatal Slave 2 PPA2 not ok', Param1 := (Set:=0, SetMin:=0, SetMax:=0,Comment:=''), Param2 := (Set:=0, SetMin:=0, SetMax:=0,Comment:='') ),
( sName := 'a_bNoCommunicationToPLCFromSlave3PPAMaster2', sClearName := '', sID := '4074', a := FALSE, b := FALSE, iGroup :=4, iSetDelay :=0, iResetDelay := 0, eResetMode := MANU, eBrakeProgram := B99, eAlarmProgram := 0, Enable := TRUE, iRepetitionNumber := 0 , iRepetitionPeriod := 0, Comment := '', Param1 := (Set:=0, SetMin:=0, SetMax:=0,Comment:=''), Param2 := (Set:=0, SetMin:=0, SetMax:=0,Comment:='') ),
( sName := 'a_bNoCommunicationToPLCFromSlave4PPAMaster3', sClearName := '', sID := '4075', a := FALSE, b := FALSE, iGroup :=4, iSetDelay :=0, iResetDelay := 0, eResetMode := MANU, eBrakeProgram := B99, eAlarmProgram := 0, Enable := TRUE, iRepetitionNumber := 0 , iRepetitionPeriod := 0, Comment := '', Param1 := (Set:=0, SetMin:=0, SetMax:=0,Comment:=''), Param2 := (Set:=0, SetMin:=0, SetMax:=0,Comment:='') ),
( sName := 'a_bNotReadyToOperate', sClearName := '', sID := '4076', a := FALSE, b := FALSE, iGroup :=4, iSetDelay :=0, iResetDelay := 0, eResetMode := MANU, eBrakeProgram := B99, eAlarmProgram := 0, Enable := TRUE, iRepetitionNumber := 0 , iRepetitionPeriod := 0, Comment := '', Param1 := (Set:=0, SetMin:=0, SetMax:=0,Comment:=''), Param2 := (Set:=0, SetMin:=0, SetMax:=0,Comment:='') ),
( sName := 'a_bPitchEncodersDisagreeSSB_Safety', sClearName := 'Encoders readings differ with SSB derived blade measurements above acceptable thresholds', sID := '4062', a := FALSE, b := FALSE, iGroup :=4, iSetDelay :=1, iResetDelay := 1, eResetMode := MANU, eBrakeProgram := B4, eAlarmProgram := 0, Enable := TRUE, iRepetitionNumber := 0 , iRepetitionPeriod := 0, Comment := 'Encoders readings differ with SSB derived blade measurements more than acceptable thresholds. Trip safety circuit.', Param1 := (Set:=3, SetMin:=3, SetMax:=3,Comment:='Degs'), Param2 := (Set:=1, SetMin:=1, SetMax:=1,Comment:='Degs') ),
( sName := 'a_bPitchEncodersDisagreeSSB_Fault', sClearName := 'Encoders readings differ with SSB derived blade measurements above acceptable thresholds', sID := '4063', a := FALSE, b := FALSE, iGroup :=4, iSetDelay :=1, iResetDelay := 1, eResetMode := MANU, eBrakeProgram := B20, eAlarmProgram := 0, Enable := TRUE, iRepetitionNumber := 0 , iRepetitionPeriod := 0, Comment := 'Encoders readings differ with SSB derived blade measurements more than acceptable thresholds. Initiate controlled shutdown.', Param1 := (Set:=1.99999971123577, SetMin:=1.99999971123577, SetMax:=1.99999971123577,Comment:='Degs'), Param2 := (Set:=1, SetMin:=1, SetMax:=1,Comment:='Degs') ),
( sName := 'a_bPitchEncodersDisagreeSSB_Warning', sClearName := 'Encoders readings differ with SSB derived blade measurements above acceptable thresholds', sID := '4064', a := FALSE, b := FALSE, iGroup :=4, iSetDelay :=1, iResetDelay := 1, eResetMode := MANU, eBrakeProgram := B99, eAlarmProgram := 0, Enable := TRUE, iRepetitionNumber := 0 , iRepetitionPeriod := 0, Comment := 'Encoders readings differ with SSB derived blade measurements more than acceptable thresholds. Notify operator', Param1 := (Set:=1.5, SetMin:=1.5, SetMax:=1.5,Comment:='Degs'), Param2 := (Set:=1, SetMin:=1, SetMax:=1,Comment:='Degs') ),
( sName := 'a_bPitchTorqueAv1sHiWarn', sClearName := 'Higher than normal torque spikes on active SSB drive warning', sID := '4080', a := FALSE, b := FALSE, iGroup :=4, iSetDelay :=1, iResetDelay := 1, eResetMode := MANU, eBrakeProgram := B99, eAlarmProgram := 0, Enable := TRUE, iRepetitionNumber := 0 , iRepetitionPeriod := 0, Comment := 'Higher than normal torque spikes on active SSB drive warning', Param1 := (Set:=300, SetMin:=0, SetMax:=320,Comment:=''), Param2 := (Set:=100, SetMin:=0, SetMax:=100,Comment:='') ),
( sName := 'a_bPitchTorqueAv1sHiAlarm', sClearName := 'Higher than normal torque spikes on active SSB drive alarm', sID := '4081', a := FALSE, b := FALSE, iGroup :=4, iSetDelay :=1, iResetDelay := 1, eResetMode := MANU, eBrakeProgram := B20, eAlarmProgram := 0, Enable := TRUE, iRepetitionNumber := 0 , iRepetitionPeriod := 0, Comment := 'Higher than normal torque spikes on active SSB drive alarm', Param1 := (Set:=320, SetMin:=0, SetMax:=320,Comment:=''), Param2 := (Set:=100, SetMin:=0, SetMax:=100,Comment:='') ),
( sName := 'a_bPitchTorqueAv5sTorqueHiWarn', sClearName := 'Higher than normal steady state torques on active SSB drive warning', sID := '4082', a := FALSE, b := FALSE, iGroup :=4, iSetDelay :=1, iResetDelay := 1, eResetMode := MANU, eBrakeProgram := B99, eAlarmProgram := 0, Enable := TRUE, iRepetitionNumber := 0 , iRepetitionPeriod := 0, Comment := 'Higher than normal steady state torques on active SSB drive', Param1 := (Set:=320, SetMin:=0, SetMax:=320,Comment:=''), Param2 := (Set:=100, SetMin:=0, SetMax:=100,Comment:='') ),
( sName := 'a_bPitchTorqueAv60sTorqueHiWarn', sClearName := 'Higher than normal average torque levels seen on SSB system warning', sID := '4083', a := FALSE, b := FALSE, iGroup :=4, iSetDelay :=1, iResetDelay := 1, eResetMode := MANU, eBrakeProgram := B99, eAlarmProgram := 0, Enable := TRUE, iRepetitionNumber := 0 , iRepetitionPeriod := 0, Comment := 'Higher than normal average torque levels seen on SSB system', Param1 := (Set:=320, SetMin:=0, SetMax:=320,Comment:=''), Param2 := (Set:=100, SetMin:=0, SetMax:=100,Comment:='') ),
( sName := 'a_bPitchDiffInStopPos', sClearName := 'Difference in pitch and feather STOP position. ', sID := '4084', a := FALSE, b := FALSE, iGroup :=4, iSetDelay :=1, iResetDelay := 1, eResetMode := MANU, eBrakeProgram := B99, eAlarmProgram := 0, Enable := TRUE, iRepetitionNumber := 0 , iRepetitionPeriod := 0, Comment := 'Difference in pitch and feather STOP position. ', Param1 := (Set:=0.4, SetMin:=0, SetMax:=2,Comment:=''), Param2 := (Set:=0.2, SetMin:=0, SetMax:=0.2,Comment:='') ),
( sName := 'a_bPitchMaxMotorTorqueExceeded', sClearName := 'Pitch Max motor torque exceeded', sID := '4085', a := FALSE, b := FALSE, iGroup :=4, iSetDelay :=1, iResetDelay := 1, eResetMode := MANU, eBrakeProgram := B20, eAlarmProgram := 0, Enable := TRUE, iRepetitionNumber := 0 , iRepetitionPeriod := 0, Comment := 'Pitch Max motor torque exceeded', Param1 := (Set:=320, SetMin:=0, SetMax:=350,Comment:='Pitch Max motor torque exceeded'), Param2 := (Set:=100, SetMin:=0, SetMax:=100,Comment:='') ),
( sName := 'a_bPitchMaxMotorCurrentExceeded', sClearName := 'Pitch Max motor current exceeded', sID := '4086', a := FALSE, b := FALSE, iGroup :=4, iSetDelay :=1, iResetDelay := 1, eResetMode := MANU, eBrakeProgram := B20, eAlarmProgram := 0, Enable := TRUE, iRepetitionNumber := 0 , iRepetitionPeriod := 0, Comment := 'Pitch Max motor current exceeded', Param1 := (Set:=70, SetMin:=28, SetMax:=80,Comment:='Pitch Max motor current exceeded'), Param2 := (Set:=19, SetMin:=0, SetMax:=20,Comment:='') ),
( sName := 'a_bPitchTrackingFault', sClearName := 'Pitch tracking fault', sID := '4087', a := FALSE, b := FALSE, iGroup :=4, iSetDelay :=10, iResetDelay := 10, eResetMode := MANU, eBrakeProgram := B20, eAlarmProgram := EMAIL, Enable := TRUE, iRepetitionNumber := 0 , iRepetitionPeriod := 10, Comment := 'Pitch tracking fault', Param1 := (Set:=2.5, SetMin:=1, SetMax:=5,Comment:=''), Param2 := (Set:=0, SetMin:=0, SetMax:=0,Comment:='') ),
( sName := 'a_bPitchTrackingWarning', sClearName := 'Pitch tracking warning', sID := '4088', a := FALSE, b := FALSE, iGroup :=4, iSetDelay :=10, iResetDelay := 10, eResetMode := MANU, eBrakeProgram := B99, eAlarmProgram := EMAIL, Enable := TRUE, iRepetitionNumber := 0 , iRepetitionPeriod := 10, Comment := 'Pitch tracking warning', Param1 := (Set:=1.5, SetMin:=1, SetMax:=3,Comment:=''), Param2 := (Set:=0, SetMin:=0, SetMax:=0,Comment:='') ),
( sName := 'a_bPitchFineSoftwareLimitSwitch', sClearName := 'Pitch system detected fine limit', sID := '4089', a := FALSE, b := FALSE, iGroup :=4, iSetDelay :=1, iResetDelay := 10, eResetMode := MANU, eBrakeProgram := B4, eAlarmProgram := 0, Enable := TRUE, iRepetitionNumber := 0 , iRepetitionPeriod := 10, Comment := 'Pitch system detected fine limit', Param1 := (Set:=-1, SetMin:=-1, SetMax:=180,Comment:=''), Param2 := (Set:=4, SetMin:=1, SetMax:=75,Comment:='') ),
